LIN {X 59.447,Y -46.624,Z -151.820,A -90.000,B 90.000,C 0.000} C_DIS
LIN {X 59.979,Y -46.636,Z -152.039,A -90.000,B 90.000,C 0.000} C_DIS
LIN {X 60.285,Y -46.643,Z -152.174,A -90.000,B 90.000,C 0.000} C_DIS
LIN {X 60.366,Y -46.645,Z -152.210,A -90.000,B 90.000,C 0.000} C_DIS
LIN {X 60.866,Y -46.657,Z -152.447,A -90.000,B 90.000,C 0.000} C_DIS
LIN {X 60.967,Y -46.654,Z -152.497,A -90.000,B 90.000,C 0.000} C_DIS
LIN {X 61.302,Y -46.635,Z -152.670,A -90.000,B 90.000,C 0.000} C_DIS
LIN {X 61.532,Y -46.619,Z -152.790,A -90.000,B 90.000,C 0.000} C_DIS
LIN {X 62.046,Y -46.587,Z -153.082,A -90.000,B 90.000,C 0.000} C_DIS
LIN {X 62.540,Y -46.557,Z -153.378,A -90.000,B 90.000,C 0.000} C_DIS
LIN {X 63.037,Y -46.527,Z -153.694,A -90.000,B 90.000,C 0.000} C_DIS
LIN {X 63.620,Y -46.494,Z -154.093,A -90.000,B 90.000,C 0.000} C_DIS
LIN {X 63.900,Y -46.478,Z -154.298,A -90.000,B 90.000,C 0.000} C_DIS
LIN {X 64.036,Y -46.460,Z -154.399,A -90.000,B 90.000,C 0.000} C_DIS
LIN {X 64.158,Y -46.443,Z -154.491,A -90.000,B 90.000,C 0.000} C_DIS
LIN {X 64.675,Y -46.369,Z -154.905,A -90.000,B 90.000,C 0.000} C_DIS
LIN {X 65.187,Y -46.297,Z -155.342,A -90.000,B 90.000,C 0.000} C_DIS
LIN {X 65.521,Y -46.250,Z -155.645,A -90.000,B 90.000,C 0.000} C_DIS
LIN {X 66.029,Y -46.178,Z -156.130,A -90.000,B 90.000,C 0.000} C_DIS
LIN {X 66.453,Y -46.120,Z -156.565,A -90.000,B 90.000,C 0.000} C_DIS
LIN {X 66.624,Y -46.096,Z -156.751,A -90.000,B 90.000,C 0.000} C_DIS
LIN {X 66.971,Y -46.029,Z -157.134,A -90.000,B 90.000,C 0.000} C_DIS
LIN {X 67.241,Y -45.966,Z -157.456,A -90.000,B 90.000,C 0.000} C_DIS
LIN {X 67.519,Y -45.898,Z -157.794,A -90.000,B 90.000,C 0.000} C_DIS
LIN {X 67.718,Y -45.848,Z -158.052,A -90.000,B 90.000,C 0.000} C_DIS
LIN {X 68.044,Y -45.766,Z -158.488,A -90.000,B 90.000,C 0.000} C_DIS
LIN {X 68.258,Y -45.712,Z -158.793,A -90.000,B 90.000,C 0.000} C_DIS
LIN {X 68.440,Y -45.666,Z -159.058,A -90.000,B 90.000,C 0.000} C_DIS
LIN {X 68.717,Y -45.595,Z -159.479,A -90.000,B 90.000,C 0.000} C_DIS
LIN {X 68.978,Y -45.527,Z -159.906,A -90.000,B 90.000,C 0.000} C_DIS
LIN {X 69.258,Y -45.454,Z -160.385,A -90.000,B 90.000,C 0.000} C_DIS
LIN {X 69.508,Y -45.387,Z -160.840,A -90.000,B 90.000,C 0.000} C_DIS
LIN {X 69.580,Y -45.368,Z -160.980,A -90.000,B 90.000,C 0.000} C_DIS
LIN {X 69.738,Y -45.308,Z -161.295,A -90.000,B 90.000,C 0.000} C_DIS
LIN {X 69.738,Y -60.000,Z -161.295,A -90.000,B 90.000,C 0.000} C_DIS
LIN {X 51.420,Y -60.000,Z -148.529,A -90.000,B 90.000,C 0.000} C_DIS
LIN {X 51.420,Y -45.308,Z -148.529,A -90.000,B 90.000,C 0.000} C_DIS
LIN {X 51.656,Y -45.359,Z -148.518,A -90.000,B 90.000,C 0.000} C_DIS
LIN {X 52.314,Y -45.502,Z -148.497,A -90.000,B 90.000,C 0.000} C_DIS
LIN {X 52.905,Y -45.633,Z -148.497,A -90.000,B 90.000,C 0.000} C_DIS
LIN {X 53.199,Y -45.699,Z -148.504,A -90.000,B 90.000,C 0.000} C_DIS
LIN {X 53.580,Y -45.759,Z -148.519,A -90.000,B 90.000,C 0.000} C_DIS
LIN {X 54.008,Y -45.829,Z -148.547,A -90.000,B 90.000,C 0.000} C_DIS
LIN {X 54.649,Y -45.936,Z -148.604,A -90.000,B 90.000,C 0.000} C_DIS
LIN {X 55.130,Y -46.016,Z -148.659,A -90.000,B 90.000,C 0.000} C_DIS
LIN {X 55.563,Y -46.087,Z -148.721,A -90.000,B 90.000,C 0.000} C_DIS
LIN {X 55.943,Y -46.141,Z -148.778,A -90.000,B 90.000,C 0.000} C_DIS
LIN {X 56.047,Y -46.155,Z -148.796,A -90.000,B 90.000,C 0.000} C_DIS
LIN {X 56.497,Y -46.195,Z -148.882,A -90.000,B 90.000,C 0.000} C_DIS
LIN {X 56.661,Y -46.209,Z -148.915,A -90.000,B 90.000,C 0.000} C_DIS
LIN {X 57.300,Y -46.275,Z -149.058,A -90.000,B 90.000,C 0.000} C_DIS
LIN {X 57.950,Y -46.344,Z -149.225,A -90.000,B 90.000,C 0.000} C_DIS
LIN {X 58.439,Y -46.397,Z -149.362,A -90.000,B 90.000,C 0.000} C_DIS
LIN {X 58.552,Y -46.409,Z -149.396,A -90.000,B 90.000,C 0.000} C_DIS
LIN {X 58.696,Y -46.417,Z -149.440,A -90.000,B 90.000,C 0.000} C_DIS
LIN {X 59.080,Y -46.425,Z -149.568,A -90.000,B 90.000,C 0.000} C_DIS
LIN {X 59.564,Y -46.434,Z -149.734,A -90.000,B 90.000,C 0.000} C_DIS
LIN {X 59.994,Y -46.444,Z -149.897,A -90.000,B 90.000,C 0.000} C_DIS
LIN {X 60.209,Y -46.450,Z -149.979,A -90.000,B 90.000,C 0.000} C_DIS
LIN {X 60.788,Y -46.470,Z -150.217,A -90.000,B 90.000,C 0.000} C_DIS
LIN {X 61.149,Y -46.483,Z -150.377,A -90.000,B 90.000,C 0.000} C_DIS
LIN {X 61.348,Y -46.491,Z -150.469,A -90.000,B 90.000,C 0.000} C_DIS
LIN {X 61.461,Y -46.494,Z -150.522,A -90.000,B 90.000,C 0.000} C_DIS
LIN {X 61.703,Y -46.490,Z -150.638,A -90.000,B 90.000,C 0.000} C_DIS
LIN {X 61.873,Y -46.482,Z -150.723,A -90.000,B 90.000,C 0.000} C_DIS
LIN {X 62.480,Y -46.449,Z -151.038,A -90.000,B 90.000,C 0.000} C_DIS
LIN {X 63.064,Y -46.419,Z -151.368,A -90.000,B 90.000,C 0.000} C_DIS
LIN {X 63.602,Y -46.393,Z -151.691,A -90.000,B 90.000,C 0.000} C_DIS
LIN {X 64.157,Y -46.368,Z -152.044,A -90.000,B 90.000,C 0.000} C_DIS
LIN {X 64.418,Y -46.358,Z -152.222,A -90.000,B 90.000,C 0.000} C_DIS
LIN {X 64.519,Y -46.351,Z -152.292,A -90.000,B 90.000,C 0.000} C_DIS
LIN {X 64.794,Y -46.316,Z -152.483,A -90.000,B 90.000,C 0.000} C_DIS
LIN {X 65.364,Y -46.243,Z -152.908,A -90.000,B 90.000,C 0.000} C_DIS
LIN {X 65.919,Y -46.170,Z -153.351,A -90.000,B 90.000,C 0.000} C_DIS
LIN {X 66.508,Y -46.088,Z -153.855,A -90.000,B 90.000,C 0.000} C_DIS
LIN {X 66.878,Y -46.036,Z -154.192,A -90.000,B 90.000,C 0.000} C_DIS
LIN {X 67.263,Y -45.983,Z -154.559,A -90.000,B 90.000,C 0.000} C_DIS
LIN {X 67.435,Y -45.949,Z -154.726,A -90.000,B 90.000,C 0.000} C_DIS
LIN {X 67.634,Y -45.911,Z -154.932,A -90.000,B 90.000,C 0.000} C_DIS
LIN {X 67.855,Y -45.862,Z -155.162,A -90.000,B 90.000,C 0.000} C_DIS
LIN {X 68.412,Y -45.738,Z -155.778,A -90.000,B 90.000,C 0.000} C_DIS
LIN {X 68.813,Y -45.649,Z -156.256,A -90.000,B 90.000,C 0.000} C_DIS
LIN {X 69.057,Y -45.594,Z -156.552,A -90.000,B 90.000,C 0.000} C_DIS
LIN {X 69.379,Y -45.522,Z -156.972,A -90.000,B 90.000,C 0.000} C_DIS
LIN {X 69.631,Y -45.465,Z -157.308,A -90.000,B 90.000,C 0.000} C_DIS
LIN {X 69.887,Y -45.407,Z -157.672,A -90.000,B 90.000,C 0.000} C_DIS
LIN {X 70.069,Y -45.363,Z -157.937,A -90.000,B 90.000,C 0.000} C_DIS
LIN {X 70.283,Y -45.308,Z -158.263,A -90.000,B 90.000,C 0.000} C_DIS
LIN {X 70.283,Y -60.000,Z -158.263,A -90.000,B 90.000,C 0.000} C_DIS
LIN {X 53.285,Y -60.000,Z -146.544,A -90.000,B 90.000,C 0.000} C_DIS
LIN {X 53.285,Y -45.308,Z -146.544,A -90.000,B 90.000,C 0.000} C_DIS
LIN {X 53.566,Y -45.372,Z -146.551,A -90.000,B 90.000,C 0.000} C_DIS
LIN {X 53.798,Y -45.420,Z -146.559,A -90.000,B 90.000,C 0.000} C_DIS
LIN {X 53.933,Y -45.449,Z -146.567,A -90.000,B 90.000,C 0.000} C_DIS
LIN {X 54.248,Y -45.505,Z -146.588,A -90.000,B 90.000,C 0.000} C_DIS
LIN {X 54.708,Y -45.588,Z -146.628,A -90.000,B 90.000,C 0.000} C_DIS
LIN {X 54.923,Y -45.624,Z -146.648,A -90.000,B 90.000,C 0.000} C_DIS
LIN {X 55.458,Y -45.716,Z -146.709,A -90.000,B 90.000,C 0.000} C_DIS
LIN {X 56.327,Y -45.869,Z -146.834,A -90.000,B 90.000,C 0.000} C_DIS
LIN {X 56.403,Y -45.881,Z -146.847,A -90.000,B 90.000,C 0.000} C_DIS
LIN {X 56.867,Y -45.935,Z -146.934,A -90.000,B 90.000,C 0.000} C_DIS
LIN {X 57.119,Y -45.961,Z -146.984,A -90.000,B 90.000,C 0.000} C_DIS
LIN {X 57.818,Y -46.036,Z -147.141,A -90.000,B 90.000,C 0.000} C_DIS
LIN {X 58.513,Y -46.115,Z -147.319,A -90.000,B 90.000,C 0.000} C_DIS
LIN {X 59.083,Y -46.192,Z -147.479,A -90.000,B 90.000,C 0.000} C_DIS
LIN {X 59.198,Y -46.208,Z -147.513,A -90.000,B 90.000,C 0.000} C_DIS
LIN {X 59.344,Y -46.218,Z -147.558,A -90.000,B 90.000,C 0.000} C_DIS
LIN {X 59.731,Y -46.232,Z -147.686,A -90.000,B 90.000,C 0.000} C_DIS
LIN {X 60.273,Y -46.252,Z -147.873,A -90.000,B 90.000,C 0.000} C_DIS
LIN {X 60.972,Y -46.281,Z -148.138,A -90.000,B 90.000,C 0.000} C_DIS
LIN {X 61.600,Y -46.310,Z -148.396,A -90.000,B 90.000,C 0.000} C_DIS
LIN {X 61.987,Y -46.328,Z -148.568,A -90.000,B 90.000,C 0.000} C_DIS
LIN {X 62.168,Y -46.329,Z -148.652,A -90.000,B 90.000,C 0.000} C_DIS
LIN {X 62.338,Y -46.325,Z -148.733,A -90.000,B 90.000,C 0.000} C_DIS
LIN {X 62.588,Y -46.314,Z -148.853,A -90.000,B 90.000,C 0.000} C_DIS
LIN {X 62.784,Y -46.305,Z -148.951,A -90.000,B 90.000,C 0.000} C_DIS
LIN {X 62.929,Y -46.298,Z -149.026,A -90.000,B 90.000,C 0.000} C_DIS
LIN {X 63.454,Y -46.274,Z -149.300,A -90.000,B 90.000,C 0.000} C_DIS
LIN {X 64.083,Y -46.246,Z -149.656,A -90.000,B 90.000,C 0.000} C_DIS
LIN {X 64.667,Y -46.221,Z -150.007,A -90.000,B 90.000,C 0.000} C_DIS
LIN {X 65.039,Y -46.205,Z -150.244,A -90.000,B 90.000,C 0.000} C_DIS
LIN {X 65.111,Y -46.200,Z -150.290,A -90.000,B 90.000,C 0.000} C_DIS
LIN {X 65.274,Y -46.179,Z -150.396,A -90.000,B 90.000,C 0.000} C_DIS
LIN {X 65.963,Y -46.090,Z -150.876,A -90.000,B 90.000,C 0.000} C_DIS
LIN {X 66.585,Y -46.011,Z -151.341,A -90.000,B 90.000,C 0.000} C_DIS
LIN {X 67.191,Y -45.937,Z -151.825,A -90.000,B 90.000,C 0.000} C_DIS
LIN {X 67.828,Y -45.860,Z -152.369,A -90.000,B 90.000,C 0.000} C_DIS
LIN {X 68.251,Y -45.787,Z -152.758,A -90.000,B 90.000,C 0.000} C_DIS
LIN {X 68.759,Y -45.683,Z -153.251,A -90.000,B 90.000,C 0.000} C_DIS
LIN {X 68.852,Y -45.664,Z -153.343,A -90.000,B 90.000,C 0.000} C_DIS
LIN {X 69.222,Y -45.588,Z -153.728,A -90.000,B 90.000,C 0.000} C_DIS
LIN {X 69.305,Y -45.570,Z -153.815,A -90.000,B 90.000,C 0.000} C_DIS
LIN {X 69.898,Y -45.438,Z -154.474,A -90.000,B 90.000,C 0.000} C_DIS
LIN {X 70.312,Y -45.346,Z -154.966,A -90.000,B 90.000,C 0.000} C_DIS
LIN {X 70.480,Y -45.308,Z -155.171,A -90.000,B 90.000,C 0.000} C_DIS
LIN {X 70.480,Y -60.000,Z -155.171,A -90.000,B 90.000,C 0.000} C_DIS
LIN {X 55.397,Y -60.000,Z -144.721,A -90.000,B 90.000,C 0.000} C_DIS
LIN {X 55.397,Y -45.308,Z -144.721,A -90.000,B 90.000,C 0.000} C_DIS
LIN {X 55.811,Y -45.386,Z -144.768,A -90.000,B 90.000,C 0.000} C_DIS
LIN {X 56.720,Y -45.560,Z -144.897,A -90.000,B 90.000,C 0.000} C_DIS
LIN {X 57.059,Y -45.621,Z -144.957,A -90.000,B 90.000,C 0.000} C_DIS
LIN {X 57.528,Y -45.677,Z -145.047,A -90.000,B 90.000,C 0.000} C_DIS
LIN {X 57.647,Y -45.689,Z -145.073,A -90.000,B 90.000,C 0.000} C_DIS
LIN {X 58.339,Y -45.777,Z -145.227,A -90.000,B 90.000,C 0.000} C_DIS
LIN {X 59.096,Y -45.878,Z -145.421,A -90.000,B 90.000,C 0.000} C_DIS
LIN {X 59.727,Y -45.963,Z -145.598,A -90.000,B 90.000,C 0.000} C_DIS
LIN {X 59.823,Y -45.976,Z -145.627,A -90.000,B 90.000,C 0.000} C_DIS
LIN {X 59.969,Y -45.987,Z -145.672,A -90.000,B 90.000,C 0.000} C_DIS
LIN {X 60.421,Y -46.003,Z -145.823,A -90.000,B 90.000,C 0.000} C_DIS
LIN {X 60.636,Y -46.011,Z -145.897,A -90.000,B 90.000,C 0.000} C_DIS
LIN {X 60.986,Y -46.030,Z -146.017,A -90.000,B 90.000,C 0.000} C_DIS
LIN {X 61.738,Y -46.074,Z -146.302,A -90.000,B 90.000,C 0.000} C_DIS
LIN {X 62.412,Y -46.116,Z -146.579,A -90.000,B 90.000,C 0.000} C_DIS
LIN {X 62.556,Y -46.122,Z -146.643,A -90.000,B 90.000,C 0.000} C_DIS
LIN {X 62.721,Y -46.124,Z -146.716,A -90.000,B 90.000,C 0.000} C_DIS
LIN {X 62.878,Y -46.121,Z -146.788,A -90.000,B 90.000,C 0.000} C_DIS
LIN {X 63.515,Y -46.097,Z -147.094,A -90.000,B 90.000,C 0.000} C_DIS
LIN {X 63.692,Y -46.091,Z -147.182,A -90.000,B 90.000,C 0.000} C_DIS
LIN {X 64.428,Y -46.066,Z -147.565,A -90.000,B 90.000,C 0.000} C_DIS
LIN {X 65.103,Y -46.053,Z -147.946,A -90.000,B 90.000,C 0.000} C_DIS
LIN {X 65.440,Y -46.047,Z -148.148,A -90.000,B 90.000,C 0.000} C_DIS
LIN {X 65.570,Y -46.042,Z -148.226,A -90.000,B 90.000,C 0.000} C_DIS
LIN {X 65.702,Y -46.029,Z -148.306,A -90.000,B 90.000,C 0.000} C_DIS
LIN {X 66.341,Y -45.956,Z -148.719,A -90.000,B 90.000,C 0.000} C_DIS
LIN {X 67.136,Y -45.868,Z -149.271,A -90.000,B 90.000,C 0.000} C_DIS
LIN {X 67.565,Y -45.821,Z -149.592,A -90.000,B 90.000,C 0.000} C_DIS
LIN {X 67.809,Y -45.791,Z -149.775,A -90.000,B 90.000,C 0.000} C_DIS
LIN {X 68.439,Y -45.713,Z -150.279,A -90.000,B 90.000,C 0.000} C_DIS
LIN {X 68.852,Y -45.639,Z -150.635,A -90.000,B 90.000,C 0.000} C_DIS
LIN {X 69.142,Y -45.580,Z -150.888,A -90.000,B 90.000,C 0.000} C_DIS
LIN {X 69.595,Y -45.487,Z -151.308,A -90.000,B 90.000,C 0.000} C_DIS
LIN {X 70.122,Y -45.379,Z -151.819,A -90.000,B 90.000,C 0.000} C_DIS
LIN {X 70.295,Y -45.344,Z -151.995,A -90.000,B 90.000,C 0.000} C_DIS
LIN {X 70.471,Y -45.308,Z -152.177,A -90.000,B 90.000,C 0.000} C_DIS
LIN {X 70.471,Y -60.000,Z -152.177,A -90.000,B 90.000,C 0.000} C_DIS
LIN {X 57.673,Y -60.000,Z -143.068,A -90.000,B 90.000,C 0.000} C_DIS
LIN {X 57.673,Y -45.308,Z -143.068,A -90.000,B 90.000,C 0.000} C_DIS
LIN {X 57.981,Y -45.358,Z -143.125,A -90.000,B 90.000,C 0.000} C_DIS
LIN {X 58.562,Y -45.455,Z -143.250,A -90.000,B 90.000,C 0.000} C_DIS
LIN {X 58.857,Y -45.494,Z -143.316,A -90.000,B 90.000,C 0.000} C_DIS
LIN {X 59.667,Y -45.605,Z -143.524,A -90.000,B 90.000,C 0.000} C_DIS
LIN {X 60.166,Y -45.674,Z -143.664,A -90.000,B 90.000,C 0.000} C_DIS
LIN {X 60.407,Y -45.704,Z -143.734,A -90.000,B 90.000,C 0.000} C_DIS
LIN {X 60.688,Y -45.731,Z -143.821,A -90.000,B 90.000,C 0.000} C_DIS
LIN {X 61.226,Y -45.785,Z -143.998,A -90.000,B 90.000,C 0.000} C_DIS
LIN {X 61.701,Y -45.815,Z -144.162,A -90.000,B 90.000,C 0.000} C_DIS
LIN {X 62.505,Y -45.867,Z -144.467,A -90.000,B 90.000,C 0.000} C_DIS
LIN {X 62.948,Y -45.898,Z -144.648,A -90.000,B 90.000,C 0.000} C_DIS
LIN {X 63.151,Y -45.907,Z -144.732,A -90.000,B 90.000,C 0.000} C_DIS
LIN {X 63.524,Y -45.912,Z -144.897,A -90.000,B 90.000,C 0.000} C_DIS
LIN {X 63.817,Y -45.906,Z -145.033,A -90.000,B 90.000,C 0.000} C_DIS
LIN {X 64.402,Y -45.896,Z -145.312,A -90.000,B 90.000,C 0.000} C_DIS
LIN {X 64.615,Y -45.892,Z -145.419,A -90.000,B 90.000,C 0.000} C_DIS
LIN {X 65.404,Y -45.875,Z -145.830,A -90.000,B 90.000,C 0.000} C_DIS
LIN {X 65.989,Y -45.864,Z -146.160,A -90.000,B 90.000,C 0.000} C_DIS
LIN {X 66.114,Y -45.858,Z -146.231,A -90.000,B 90.000,C 0.000} C_DIS
LIN {X 66.199,Y -45.850,Z -146.283,A -90.000,B 90.000,C 0.000} C_DIS
LIN {X 66.754,Y -45.786,Z -146.623,A -90.000,B 90.000,C 0.000} C_DIS
LIN {X 67.454,Y -45.711,Z -147.076,A -90.000,B 90.000,C 0.000} C_DIS
LIN {X 67.702,Y -45.686,Z -147.248,A -90.000,B 90.000,C 0.000} C_DIS
LIN {X 68.305,Y -45.623,Z -147.667,A -90.000,B 90.000,C 0.000} C_DIS
LIN {X 68.893,Y -45.563,Z -148.106,A -90.000,B 90.000,C 0.000} C_DIS
LIN {X 69.052,Y -45.538,Z -148.229,A -90.000,B 90.000,C 0.000} C_DIS
LIN {X 69.317,Y -45.495,Z -148.442,A -90.000,B 90.000,C 0.000} C_DIS
LIN {X 69.700,Y -45.422,Z -148.754,A -90.000,B 90.000,C 0.000} C_DIS
LIN {X 70.298,Y -45.308,Z -149.272,A -90.000,B 90.000,C 0.000} C_DIS
LIN {X 70.298,Y -60.000,Z -149.272,A -90.000,B 90.000,C 0.000} C_DIS
LIN {X 60.225,Y -60.000,Z -141.626,A -90.000,B 90.000,C 0.000} C_DIS
LIN {X 60.225,Y -45.308,Z -141.626,A -90.000,B 90.000,C 0.000} C_DIS
LIN {X 60.347,Y -45.329,Z -141.660,A -90.000,B 90.000,C 0.000} C_DIS
LIN {X 60.767,Y -45.387,Z -141.778,A -90.000,B 90.000,C 0.000} C_DIS
LIN {X 60.971,Y -45.412,Z -141.837,A -90.000,B 90.000,C 0.000} C_DIS
LIN {X 61.330,Y -45.447,Z -141.949,A -90.000,B 90.000,C 0.000} C_DIS
LIN {X 61.949,Y -45.509,Z -142.153,A -90.000,B 90.000,C 0.000} C_DIS
LIN {X 62.419,Y -45.557,Z -142.313,A -90.000,B 90.000,C 0.000} C_DIS
LIN {X 62.933,Y -45.611,Z -142.505,A -90.000,B 90.000,C 0.000} C_DIS
LIN {X 63.273,Y -45.634,Z -142.635,A -90.000,B 90.000,C 0.000} C_DIS
LIN {X 63.488,Y -45.648,Z -142.723,A -90.000,B 90.000,C 0.000} C_DIS
LIN {X 63.608,Y -45.654,Z -142.773,A -90.000,B 90.000,C 0.000} C_DIS
LIN {X 63.900,Y -45.658,Z -142.895,A -90.000,B 90.000,C 0.000} C_DIS
LIN {X 64.355,Y -45.665,Z -143.095,A -90.000,B 90.000,C 0.000} C_DIS
LIN {X 64.669,Y -45.670,Z -143.239,A -90.000,B 90.000,C 0.000} C_DIS
LIN {X 65.147,Y -45.679,Z -143.465,A -90.000,B 90.000,C 0.000} C_DIS
LIN {X 65.384,Y -45.675,Z -143.581,A -90.000,B 90.000,C 0.000} C_DIS
LIN {X 65.531,Y -45.673,Z -143.654,A -90.000,B 90.000,C 0.000} C_DIS
LIN {X 66.367,Y -45.661,Z -144.090,A -90.000,B 90.000,C 0.000} C_DIS
LIN {X 66.431,Y -45.660,Z -144.126,A -90.000,B 90.000,C 0.000} C_DIS
LIN {X 66.624,Y -45.649,Z -144.236,A -90.000,B 90.000,C 0.000} C_DIS
LIN {X 67.126,Y -45.612,Z -144.524,A -90.000,B 90.000,C 0.000} C_DIS
LIN {X 67.404,Y -45.592,Z -144.692,A -90.000,B 90.000,C 0.000} C_DIS
LIN {X 67.816,Y -45.551,Z -144.944,A -90.000,B 90.000,C 0.000} C_DIS
LIN {X 68.570,Y -45.476,Z -145.433,A -90.000,B 90.000,C 0.000} C_DIS
LIN {X 69.377,Y -45.399,Z -145.993,A -90.000,B 90.000,C 0.000} C_DIS
LIN {X 69.423,Y -45.392,Z -146.025,A -90.000,B 90.000,C 0.000} C_DIS
LIN {X 69.561,Y -45.372,Z -146.127,A -90.000,B 90.000,C 0.000} C_DIS
LIN {X 69.817,Y -45.330,Z -146.321,A -90.000,B 90.000,C 0.000} C_DIS
LIN {X 69.929,Y -45.308,Z -146.406,A -90.000,B 90.000,C 0.000} C_DIS
LIN {X 70.238,Y -45.253,Z -146.643,A -90.000,B 90.000,C 0.000} C_DIS
LIN {X 70.507,Y -45.203,Z -146.852,A -90.000,B 90.000,C 0.000} C_DIS
LIN {X 70.735,Y -45.160,Z -147.034,A -90.000,B 90.000,C 0.000} C_DIS
LIN {X 71.005,Y -45.110,Z -147.258,A -90.000,B 90.000,C 0.000} C_DIS
LIN {X 71.139,Y -45.085,Z -147.375,A -90.000,B 90.000,C 0.000} C_DIS
LIN {X 71.274,Y -45.060,Z -147.506,A -90.000,B 90.000,C 0.000} C_DIS
LIN {X 71.302,Y -45.055,Z -147.538,A -90.000,B 90.000,C 0.000} C_DIS
LIN {X 71.330,Y -45.050,Z -147.575,A -90.000,B 90.000,C 0.000} C_DIS
LIN {X 71.338,Y -45.049,Z -147.593,A -90.000,B 90.000,C 0.000} C_DIS
LIN {X 71.339,Y -45.049,Z -147.600,A -90.000,B 90.000,C 0.000} C_DIS
LIN {X 71.336,Y -45.049,Z -147.610,A -90.000,B 90.000,C 0.000} C_DIS
LIN {X 71.317,Y -45.053,Z -147.616,A -90.000,B 90.000,C 0.000} C_DIS
LIN {X 71.282,Y -45.061,Z -147.610,A -90.000,B 90.000,C 0.000} C_DIS
LIN {X 71.250,Y -45.067,Z -147.599,A -90.000,B 90.000,C 0.000} C_DIS
LIN {X 71.166,Y -45.084,Z -147.565,A -90.000,B 90.000,C 0.000} C_DIS
LIN {X 70.992,Y -45.117,Z -147.479,A -90.000,B 90.000,C 0.000} C_DIS
LIN {X 70.677,Y -45.178,Z -147.305,A -90.000,B 90.000,C 0.000} C_DIS
LIN {X 70.279,Y -45.255,Z -147.070,A -90.000,B 90.000,C 0.000} C_DIS
LIN {X 69.809,Y -45.347,Z -146.780,A -90.000,B 90.000,C 0.000} C_DIS
LIN {X 69.550,Y -45.397,Z -146.617,A -90.000,B 90.000,C 0.000} C_DIS
LIN {X 69.276,Y -45.435,Z -146.443,A -90.000,B 90.000,C 0.000} C_DIS
LIN {X 68.693,Y -45.497,Z -146.065,A -90.000,B 90.000,C 0.000} C_DIS
LIN {X 68.386,Y -45.528,Z -145.863,A -90.000,B 90.000,C 0.000} C_DIS
LIN {X 67.747,Y -45.591,Z -145.437,A -90.000,B 90.000,C 0.000} C_DIS
LIN {X 67.084,Y -45.654,Z -144.987,A -90.000,B 90.000,C 0.000} C_DIS
LIN {X 66.409,Y -45.696,Z -144.520,A -90.000,B 90.000,C 0.000} C_DIS
LIN {X 66.070,Y -45.699,Z -144.283,A -90.000,B 90.000,C 0.000} C_DIS
LIN {X 65.396,Y -45.697,Z -143.804,A -90.000,B 90.000,C 0.000} C_DIS
LIN {X 65.065,Y -45.695,Z -143.564,A -90.000,B 90.000,C 0.000} C_DIS
LIN {X 64.738,Y -45.679,Z -143.325,A -90.000,B 90.000,C 0.000} C_DIS
LIN {X 64.105,Y -45.646,Z -142.853,A -90.000,B 90.000,C 0.000} C_DIS
LIN {X 63.801,Y -45.629,Z -142.622,A -90.000,B 90.000,C 0.000} C_DIS
LIN {X 63.508,Y -45.605,Z -142.396,A -90.000,B 90.000,C 0.000} C_DIS
LIN {X 63.227,Y -45.571,Z -142.174,A -90.000,B 90.000,C 0.000} C_DIS
LIN {X 62.959,Y -45.526,Z -141.959,A -90.000,B 90.000,C 0.000} C_DIS
LIN {X 62.585,Y -45.457,Z -141.649,A -90.000,B 90.000,C 0.000} C_DIS
LIN {X 62.249,Y -45.398,Z -141.357,A -90.000,B 90.000,C 0.000} C_DIS
LIN {X 62.048,Y -45.361,Z -141.175,A -90.000,B 90.000,C 0.000} C_DIS
LIN {X 61.867,Y -45.327,Z -141.003,A -90.000,B 90.000,C 0.000} C_DIS
LIN {X 61.707,Y -45.294,Z -140.842,A -90.000,B 90.000,C 0.000} C_DIS
LIN {X 61.571,Y -45.257,Z -140.692,A -90.000,B 90.000,C 0.000} C_DIS
LIN {X 61.458,Y -45.222,Z -140.556,A -90.000,B 90.000,C 0.000} C_DIS
LIN {X 61.411,Y -45.206,Z -140.493,A -90.000,B 90.000,C 0.000} C_DIS
LIN {X 61.371,Y -45.191,Z -140.434,A -90.000,B 90.000,C 0.000} C_DIS
LIN {X 61.324,Y -45.172,Z -140.352,A -90.000,B 90.000,C 0.000} C_DIS
LIN {X 61.292,Y -45.155,Z -140.278,A -90.000,B 90.000,C 0.000} C_DIS
LIN {X 61.280,Y -45.146,Z -140.234,A -90.000,B 90.000,C 0.000} C_DIS
LIN {X 61.275,Y -45.134,Z -140.175,A -90.000,B 90.000,C 0.000} C_DIS
LIN {X 61.282,Y -45.129,Z -140.142,A -90.000,B 90.000,C 0.000} C_DIS
LIN {X 61.296,Y -45.124,Z -140.112,A -90.000,B 90.000,C 0.000} C_DIS
LIN {X 61.307,Y -45.123,Z -140.099,A -90.000,B 90.000,C 0.000} C_DIS
LIN {X 61.333,Y -45.120,Z -140.076,A -90.000,B 90.000,C 0.000} C_DIS
LIN {X 61.389,Y -45.120,Z -140.051,A -90.000,B 90.000,C 0.000} C_DIS
LIN {X 61.436,Y -45.122,Z -140.040,A -90.000,B 90.000,C 0.000} C_DIS
LIN {X 61.492,Y -45.125,Z -140.034,A -90.000,B 90.000,C 0.000} C_DIS
LIN {X 61.558,Y -45.130,Z -140.033,A -90.000,B 90.000,C 0.000} C_DIS
LIN {X 61.672,Y -45.141,Z -140.041,A -90.000,B 90.000,C 0.000} C_DIS
LIN {X 61.760,Y -45.151,Z -140.053,A -90.000,B 90.000,C 0.000} C_DIS
LIN {X 61.965,Y -45.175,Z -140.093,A -90.000,B 90.000,C 0.000} C_DIS
LIN {X 62.209,Y -45.207,Z -140.155,A -90.000,B 90.000,C 0.000} C_DIS
LIN {X 62.346,Y -45.225,Z -140.195,A -90.000,B 90.000,C 0.000} C_DIS
LIN {X 62.494,Y -45.241,Z -140.240,A -90.000,B 90.000,C 0.000} C_DIS
LIN {X 62.820,Y -45.272,Z -140.349,A -90.000,B 90.000,C 0.000} C_DIS
LIN {X 63.190,Y -45.308,Z -140.484,A -90.000,B 90.000,C 0.000} C_DIS
LIN {X 63.862,Y -45.376,Z -140.736,A -90.000,B 90.000,C 0.000} C_DIS
LIN {X 63.917,Y -45.381,Z -140.756,A -90.000,B 90.000,C 0.000} C_DIS
LIN {X 64.135,Y -45.392,Z -140.844,A -90.000,B 90.000,C 0.000} C_DIS
LIN {X 64.700,Y -45.422,Z -141.077,A -90.000,B 90.000,C 0.000} C_DIS
LIN {X 65.187,Y -45.427,Z -141.292,A -90.000,B 90.000,C 0.000} C_DIS
LIN {X 65.574,Y -45.432,Z -141.470,A -90.000,B 90.000,C 0.000} C_DIS
LIN {X 66.014,Y -45.438,Z -141.679,A -90.000,B 90.000,C 0.000} C_DIS
LIN {X 66.418,Y -45.444,Z -141.876,A -90.000,B 90.000,C 0.000} C_DIS
LIN {X 66.710,Y -45.449,Z -142.027,A -90.000,B 90.000,C 0.000} C_DIS
LIN {X 66.868,Y -45.447,Z -142.109,A -90.000,B 90.000,C 0.000} C_DIS
LIN {X 67.087,Y -45.434,Z -142.225,A -90.000,B 90.000,C 0.000} C_DIS
LIN {X 67.353,Y -45.413,Z -142.368,A -90.000,B 90.000,C 0.000} C_DIS
LIN {X 68.139,Y -45.355,Z -142.819,A -90.000,B 90.000,C 0.000} C_DIS
LIN {X 68.795,Y -45.308,Z -143.217,A -90.000,B 90.000,C 0.000} C_DIS
LIN {X 68.795,Y -60.000,Z -143.217,A -90.000,B 90.000,C 0.000} C_DIS
LIN {X 21.437,Y -60.000,Z -200.643,A -90.000,B 90.000,C 0.000} C_DIS
LIN {X 21.437,Y -45.308,Z -200.643,A -90.000,B 90.000,C 0.000} C_DIS
LIN {X 21.642,Y -45.328,Z -200.052,A -90.000,B 90.000,C 0.000} C_DIS
LIN {X 21.753,Y -45.340,Z -199.753,A -90.000,B 90.000,C 0.000} C_DIS
LIN {X 22.022,Y -45.372,Z -199.088,A -90.000,B 90.000,C 0.000} C_DIS
LIN {X 22.066,Y -45.377,Z -198.962,A -90.000,B 90.000,C 0.000} C_DIS
LIN {X 22.972,Y -45.479,Z -196.594,A -90.000,B 90.000,C 0.000} C_DIS
LIN {X 23.048,Y -45.481,Z -196.226,A -90.000,B 90.000,C 0.000} C_DIS
LIN {X 23.142,Y -45.482,Z -195.852,A -90.000,B 90.000,C 0.000} C_DIS
LIN {X 23.197,Y -45.483,Z -195.651,A -90.000,B 90.000,C 0.000} C_DIS
LIN {X 23.294,Y -45.486,Z -195.320,A -90.000,B 90.000,C 0.000} C_DIS
LIN {X 23.416,Y -45.489,Z -194.956,A -90.000,B 90.000,C 0.000} C_DIS
LIN {X 23.860,Y -45.511,Z -193.771,A -90.000,B 90.000,C 0.000} C_DIS
LIN {X 23.928,Y -45.489,Z -193.299,A -90.000,B 90.000,C 0.000} C_DIS
LIN {X 23.996,Y -45.472,Z -192.905,A -90.000,B 90.000,C 0.000} C_DIS
LIN {X 24.063,Y -45.462,Z -192.583,A -90.000,B 90.000,C 0.000} C_DIS
LIN {X 24.148,Y -45.454,Z -192.215,A -90.000,B 90.000,C 0.000} C_DIS
LIN {X 24.221,Y -45.442,Z -191.941,A -90.000,B 90.000,C 0.000} C_DIS
LIN {X 24.335,Y -45.426,Z -191.571,A -90.000,B 90.000,C 0.000} C_DIS
LIN {X 24.388,Y -45.420,Z -191.413,A -90.000,B 90.000,C 0.000} C_DIS
LIN {X 24.556,Y -45.407,Z -190.951,A -90.000,B 90.000,C 0.000} C_DIS
LIN {X 24.669,Y -45.402,Z -190.671,A -90.000,B 90.000,C 0.000} C_DIS
LIN {X 24.849,Y -45.402,Z -190.259,A -90.000,B 90.000,C 0.000} C_DIS
LIN {X 24.895,Y -45.402,Z -190.152,A -90.000,B 90.000,C 0.000} C_DIS
LIN {X 25.316,Y -45.322,Z -188.533,A -90.000,B 90.000,C 0.000} C_DIS
LIN {X 25.368,Y -45.315,Z -188.359,A -90.000,B 90.000,C 0.000} C_DIS
LIN {X 25.390,Y -45.308,Z -188.285,A -90.000,B 90.000,C 0.000} C_DIS
LIN {X 25.390,Y -60.000,Z -188.285,A -90.000,B 90.000,C 0.000} C_DIS
LIN {X 9.368,Y -60.000,Z -243.561,A -90.000,B 90.000,C 0.000} C_DIS
LIN {X 9.368,Y -46.616,Z -243.561,A -90.000,B 90.000,C 0.000} C_DIS
LIN {X 8.562,Y -46.555,Z -242.196,A -90.000,B 90.000,C 0.000} C_DIS
LIN {X 8.317,Y -46.536,Z -241.760,A -90.000,B 90.000,C 0.000} C_DIS
LIN {X 8.219,Y -46.529,Z -241.573,A -90.000,B 90.000,C 0.000} C_DIS
LIN {X 8.140,Y -46.518,Z -241.417,A -90.000,B 90.000,C 0.000} C_DIS
LIN {X 7.998,Y -46.498,Z -241.118,A -90.000,B 90.000,C 0.000} C_DIS
LIN {X 7.944,Y -46.481,Z -240.992,A -90.000,B 90.000,C 0.000} C_DIS
LIN {X 7.869,Y -46.458,Z -240.814,A -90.000,B 90.000,C 0.000} C_DIS
LIN {X 7.812,Y -46.439,Z -240.672,A -90.000,B 90.000,C 0.000} C_DIS
LIN {X 7.699,Y -46.399,Z -240.353,A -90.000,B 90.000,C 0.000} C_DIS
LIN {X 7.516,Y -46.327,Z -239.759,A -90.000,B 90.000,C 0.000} C_DIS
LIN {X 7.433,Y -46.294,Z -239.471,A -90.000,B 90.000,C 0.000} C_DIS
LIN {X 7.370,Y -46.266,Z -239.217,A -90.000,B 90.000,C 0.000} C_DIS
LIN {X 7.341,Y -46.252,Z -239.092,A -90.000,B 90.000,C 0.000} C_DIS
LIN {X 7.280,Y -46.220,Z -238.781,A -90.000,B 90.000,C 0.000} C_DIS
LIN {X 7.237,Y -46.193,Z -238.516,A -90.000,B 90.000,C 0.000} C_DIS
LIN {X 7.145,Y -46.124,Z -237.812,A -90.000,B 90.000,C 0.000} C_DIS
LIN {X 7.104,Y -46.084,Z -237.389,A -90.000,B 90.000,C 0.000} C_DIS
LIN {X 7.085,Y -46.059,Z -237.120,A -90.000,B 90.000,C 0.000} C_DIS
LIN {X 7.067,Y -46.020,Z -236.662,A -90.000,B 90.000,C 0.000} C_DIS
LIN {X 7.065,Y -46.009,Z -236.537,A -90.000,B 90.000,C 0.000} C_DIS
LIN {X 7.066,Y -45.986,Z -236.300,A -90.000,B 90.000,C 0.000} C_DIS
LIN {X 7.070,Y -45.967,Z -236.107,A -90.000,B 90.000,C 0.000} C_DIS
LIN {X 7.087,Y -45.932,Z -235.742,A -90.000,B 90.000,C 0.000} C_DIS
LIN {X 7.111,Y -45.901,Z -235.468,A -90.000,B 90.000,C 0.000} C_DIS
LIN {X 7.143,Y -45.872,Z -235.204,A -90.000,B 90.000,C 0.000} C_DIS
LIN {X 7.175,Y -45.848,Z -234.971,A -90.000,B 90.000,C 0.000} C_DIS
LIN {X 7.243,Y -45.810,Z -234.578,A -90.000,B 90.000,C 0.000} C_DIS
LIN {X 7.485,Y -45.705,Z -233.428,A -90.000,B 90.000,C 0.000} C_DIS
LIN {X 8.325,Y -45.354,Z -229.481,A -90.000,B 90.000,C 0.000} C_DIS
LIN {X 8.459,Y -45.308,Z -228.933,A -90.000,B 90.000,C 0.000} C_DIS
LIN {X 8.459,Y -60.000,Z -228.933,A -90.000,B 90.000,C 0.000} C_DIS
LIN {X 7.048,Y -60.000,Z -243.561,A -90.000,B 90.000,C 0.000} C_DIS
LIN {X 7.048,Y -46.480,Z -243.561,A -90.000,B 90.000,C 0.000} C_DIS
LIN {X 6.824,Y -46.464,Z -243.180,A -90.000,B 90.000,C 0.000} C_DIS
LIN {X 6.581,Y -46.432,Z -242.748,A -90.000,B 90.000,C 0.000} C_DIS
LIN {X 6.545,Y -46.422,Z -242.681,A -90.000,B 90.000,C 0.000} C_DIS
LIN {X 6.339,Y -46.363,Z -242.273,A -90.000,B 90.000,C 0.000} C_DIS
LIN {X 6.202,Y -46.321,Z -241.980,A -90.000,B 90.000,C 0.000} C_DIS
LIN {X 6.124,Y -46.297,Z -241.802,A -90.000,B 90.000,C 0.000} C_DIS
LIN {X 5.973,Y -46.248,Z -241.435,A -90.000,B 90.000,C 0.000} C_DIS
LIN {X 5.831,Y -46.198,Z -241.039,A -90.000,B 90.000,C 0.000} C_DIS
LIN {X 5.774,Y -46.176,Z -240.860,A -90.000,B 90.000,C 0.000} C_DIS
LIN {X 5.623,Y -46.126,Z -240.373,A -90.000,B 90.000,C 0.000} C_DIS
LIN {X 5.524,Y -46.091,Z -240.032,A -90.000,B 90.000,C 0.000} C_DIS
LIN {X 5.445,Y -46.060,Z -239.719,A -90.000,B 90.000,C 0.000} C_DIS
LIN {X 5.414,Y -46.047,Z -239.587,A -90.000,B 90.000,C 0.000} C_DIS
LIN {X 5.333,Y -46.010,Z -239.188,A -90.000,B 90.000,C 0.000} C_DIS
LIN {X 5.277,Y -45.980,Z -238.856,A -90.000,B 90.000,C 0.000} C_DIS
LIN {X 5.242,Y -45.957,Z -238.595,A -90.000,B 90.000,C 0.000} C_DIS
LIN {X 5.179,Y -45.886,Z -238.090,A -90.000,B 90.000,C 0.000} C_DIS
LIN {X 5.134,Y -45.817,Z -237.606,A -90.000,B 90.000,C 0.000} C_DIS
LIN {X 5.119,Y -45.786,Z -237.386,A -90.000,B 90.000,C 0.000} C_DIS
LIN {X 5.109,Y -45.761,Z -237.197,A -90.000,B 90.000,C 0.000} C_DIS
LIN {X 5.093,Y -45.689,Z -236.657,A -90.000,B 90.000,C 0.000} C_DIS
LIN {X 5.095,Y -45.647,Z -236.324,A -90.000,B 90.000,C 0.000} C_DIS
LIN {X 5.103,Y -45.614,Z -236.053,A -90.000,B 90.000,C 0.000} C_DIS
LIN {X 5.126,Y -45.561,Z -235.614,A -90.000,B 90.000,C 0.000} C_DIS
LIN {X 5.152,Y -45.527,Z -235.321,A -90.000,B 90.000,C 0.000} C_DIS
LIN {X 5.188,Y -45.493,Z -235.012,A -90.000,B 90.000,C 0.000} C_DIS
LIN {X 5.226,Y -45.464,Z -234.741,A -90.000,B 90.000,C 0.000} C_DIS
LIN {X 5.305,Y -45.418,Z -234.280,A -90.000,B 90.000,C 0.000} C_DIS
LIN {X 5.544,Y -45.308,Z -233.142,A -90.000,B 90.000,C 0.000} C_DIS
LIN {X 5.544,Y -60.000,Z -233.142,A -90.000,B 90.000,C 0.000} C_DIS
LIN {X 4.754,Y -60.000,Z -243.561,A -90.000,B 90.000,C 0.000} C_DIS
LIN {X 4.754,Y -46.292,Z -243.561,A -90.000,B 90.000,C 0.000} C_DIS
LIN {X 4.565,Y -46.240,Z -243.188,A -90.000,B 90.000,C 0.000} C_DIS
LIN {X 4.400,Y -46.198,Z -242.838,A -90.000,B 90.000,C 0.000} C_DIS
LIN {X 4.339,Y -46.183,Z -242.701,A -90.000,B 90.000,C 0.000} C_DIS
LIN {X 4.133,Y -46.127,Z -242.209,A -90.000,B 90.000,C 0.000} C_DIS
LIN {X 4.099,Y -46.117,Z -242.122,A -90.000,B 90.000,C 0.000} C_DIS
LIN {X 3.934,Y -46.067,Z -241.658,A -90.000,B 90.000,C 0.000} C_DIS
LIN {X 3.732,Y -46.001,Z -241.013,A -90.000,B 90.000,C 0.000} C_DIS
LIN {X 3.611,Y -45.958,Z -240.600,A -90.000,B 90.000,C 0.000} C_DIS
LIN {X 3.572,Y -45.944,Z -240.449,A -90.000,B 90.000,C 0.000} C_DIS
LIN {X 3.535,Y -45.920,Z -240.300,A -90.000,B 90.000,C 0.000} C_DIS
LIN {X 3.475,Y -45.879,Z -240.045,A -90.000,B 90.000,C 0.000} C_DIS
LIN {X 3.387,Y -45.810,Z -239.603,A -90.000,B 90.000,C 0.000} C_DIS
LIN {X 3.321,Y -45.749,Z -239.205,A -90.000,B 90.000,C 0.000} C_DIS
LIN {X 3.216,Y -45.626,Z -238.372,A -90.000,B 90.000,C 0.000} C_DIS
LIN {X 3.164,Y -45.548,Z -237.829,A -90.000,B 90.000,C 0.000} C_DIS
LIN {X 3.145,Y -45.510,Z -237.559,A -90.000,B 90.000,C 0.000} C_DIS
LIN {X 3.134,Y -45.481,Z -237.343,A -90.000,B 90.000,C 0.000} C_DIS
LIN {X 3.116,Y -45.402,Z -236.750,A -90.000,B 90.000,C 0.000} C_DIS
LIN {X 3.117,Y -45.355,Z -236.391,A -90.000,B 90.000,C 0.000} C_DIS
LIN {X 3.126,Y -45.308,Z -236.012,A -90.000,B 90.000,C 0.000} C_DIS
LIN {X 3.129,Y -45.292,Z -235.840,A -90.000,B 90.000,C 0.000} C_DIS
LIN {X 3.148,Y -45.237,Z -235.389,A -90.000,B 90.000,C 0.000} C_DIS
LIN {X 3.163,Y -45.207,Z -235.139,A -90.000,B 90.000,C 0.000} C_DIS
LIN {X 3.191,Y -45.167,Z -234.837,A -90.000,B 90.000,C 0.000} C_DIS
LIN {X 3.212,Y -45.147,Z -234.683,A -90.000,B 90.000,C 0.000} C_DIS
LIN {X 3.223,Y -45.139,Z -234.619,A -90.000,B 90.000,C 0.000} C_DIS
LIN {X 3.247,Y -45.128,Z -234.519,A -90.000,B 90.000,C 0.000} C_DIS
LIN {X 3.258,Y -45.124,Z -234.480,A -90.000,B 90.000,C 0.000} C_DIS
LIN {X 3.278,Y -45.121,Z -234.440,A -90.000,B 90.000,C 0.000} C_DIS
LIN {X 3.292,Y -45.121,Z -234.423,A -90.000,B 90.000,C 0.000} C_DIS
LIN {X 3.311,Y -45.123,Z -234.413,A -90.000,B 90.000,C 0.000} C_DIS
LIN {X 3.326,Y -45.126,Z -234.416,A -90.000,B 90.000,C 0.000} C_DIS
LIN {X 3.348,Y -45.133,Z -234.434,A -90.000,B 90.000,C 0.000} C_DIS
LIN {X 3.385,Y -45.150,Z -234.500,A -90.000,B 90.000,C 0.000} C_DIS
LIN {X 3.401,Y -45.159,Z -234.539,A -90.000,B 90.000,C 0.000} C_DIS
LIN {X 3.432,Y -45.180,Z -234.636,A -90.000,B 90.000,C 0.000} C_DIS
LIN {X 3.465,Y -45.204,Z -234.758,A -90.000,B 90.000,C 0.000} C_DIS
LIN {X 3.516,Y -45.242,Z -234.985,A -90.000,B 90.000,C 0.000} C_DIS
LIN {X 3.548,Y -45.269,Z -235.165,A -90.000,B 90.000,C 0.000} C_DIS
LIN {X 3.616,Y -45.333,Z -235.583,A -90.000,B 90.000,C 0.000} C_DIS
LIN {X 3.715,Y -45.445,Z -236.342,A -90.000,B 90.000,C 0.000} C_DIS
LIN {X 3.780,Y -45.529,Z -236.919,A -90.000,B 90.000,C 0.000} C_DIS
LIN {X 3.840,Y -45.618,Z -237.540,A -90.000,B 90.000,C 0.000} C_DIS
LIN {X 3.868,Y -45.664,Z -237.865,A -90.000,B 90.000,C 0.000} C_DIS
LIN {X 3.921,Y -45.758,Z -238.533,A -90.000,B 90.000,C 0.000} C_DIS
LIN {X 3.966,Y -45.854,Z -239.220,A -90.000,B 90.000,C 0.000} C_DIS
LIN {X 3.985,Y -45.901,Z -239.566,A -90.000,B 90.000,C 0.000} C_DIS
LIN {X 4.002,Y -45.942,Z -239.913,A -90.000,B 90.000,C 0.000} C_DIS
LIN {X 4.017,Y -45.971,Z -240.259,A -90.000,B 90.000,C 0.000} C_DIS
LIN {X 4.038,Y -46.024,Z -240.943,A -90.000,B 90.000,C 0.000} C_DIS
LIN {X 4.046,Y -46.050,Z -241.279,A -90.000,B 90.000,C 0.000} C_DIS
LIN {X 4.049,Y -46.075,Z -241.608,A -90.000,B 90.000,C 0.000} C_DIS
LIN {X 4.049,Y -46.123,Z -242.241,A -90.000,B 90.000,C 0.000} C_DIS
LIN {X 4.033,Y -46.166,Z -242.834,A -90.000,B 90.000,C 0.000} C_DIS
LIN {X 4.021,Y -46.188,Z -243.112,A -90.000,B 90.000,C 0.000} C_DIS
LIN {X 4.002,Y -46.214,Z -243.375,A -90.000,B 90.000,C 0.000} C_DIS
LIN {X 3.966,Y -46.249,Z -243.739,A -90.000,B 90.000,C 0.000} C_DIS
LIN {X 3.920,Y -46.278,Z -244.064,A -90.000,B 90.000,C 0.000} C_DIS
LIN {X 3.865,Y -46.303,Z -244.345,A -90.000,B 90.000,C 0.000} C_DIS
LIN {X 3.821,Y -46.315,Z -244.506,A -90.000,B 90.000,C 0.000} C_DIS
LIN {X 3.798,Y -46.319,Z -244.577,A -90.000,B 90.000,C 0.000} C_DIS
LIN {X 3.748,Y -46.324,Z -244.703,A -90.000,B 90.000,C 0.000} C_DIS
LIN {X 3.734,Y -46.324,Z -244.730,A -90.000,B 90.000,C 0.000} C_DIS
LIN {X 3.691,Y -46.325,Z -244.803,A -90.000,B 90.000,C 0.000} C_DIS
LIN {X 3.645,Y -46.325,Z -244.860,A -90.000,B 90.000,C 0.000} C_DIS
LIN {X 3.613,Y -46.324,Z -244.890,A -90.000,B 90.000,C 0.000} C_DIS
LIN {X 3.562,Y -46.323,Z -244.924,A -90.000,B 90.000,C 0.000} C_DIS
LIN {X 3.507,Y -46.322,Z -244.939,A -90.000,B 90.000,C 0.000} C_DIS
LIN {X 3.469,Y -46.321,Z -244.940,A -90.000,B 90.000,C 0.000} C_DIS
LIN {X 3.408,Y -46.317,Z -244.927,A -90.000,B 90.000,C 0.000} C_DIS
LIN {X 3.366,Y -46.313,Z -244.908,A -90.000,B 90.000,C 0.000} C_DIS
LIN {X 3.322,Y -46.308,Z -244.882,A -90.000,B 90.000,C 0.000} C_DIS
LIN {X 3.255,Y -46.300,Z -244.825,A -90.000,B 90.000,C 0.000} C_DIS
LIN {X 3.181,Y -46.290,Z -244.749,A -90.000,B 90.000,C 0.000} C_DIS
LIN {X 3.130,Y -46.281,Z -244.689,A -90.000,B 90.000,C 0.000} C_DIS
LIN {X 3.077,Y -46.270,Z -244.620,A -90.000,B 90.000,C 0.000} C_DIS
LIN {X 3.024,Y -46.257,Z -244.542,A -90.000,B 90.000,C 0.000} C_DIS
LIN {X 2.912,Y -46.229,Z -244.356,A -90.000,B 90.000,C 0.000} C_DIS
LIN {X 2.792,Y -46.197,Z -244.132,A -90.000,B 90.000,C 0.000} C_DIS
LIN {X 2.666,Y -46.160,Z -243.868,A -90.000,B 90.000,C 0.000} C_DIS
LIN {X 2.600,Y -46.139,Z -243.720,A -90.000,B 90.000,C 0.000} C_DIS
LIN {X 2.534,Y -46.118,Z -243.561,A -90.000,B 90.000,C 0.000} C_DIS
LIN {X 2.294,Y -46.040,Z -242.990,A -90.000,B 90.000,C 0.000} C_DIS
LIN {X 2.240,Y -46.021,Z -242.853,A -90.000,B 90.000,C 0.000} C_DIS
LIN {X 2.057,Y -45.954,Z -242.340,A -90.000,B 90.000,C 0.000} C_DIS
LIN {X 2.032,Y -45.945,Z -242.266,A -90.000,B 90.000,C 0.000} C_DIS
LIN {X 1.983,Y -45.926,Z -242.106,A -90.000,B 90.000,C 0.000} C_DIS
LIN {X 1.927,Y -45.894,Z -241.925,A -90.000,B 90.000,C 0.000} C_DIS
LIN {X 1.839,Y -45.850,Z -241.640,A -90.000,B 90.000,C 0.000} C_DIS
LIN {X 1.704,Y -45.779,Z -241.176,A -90.000,B 90.000,C 0.000} C_DIS
LIN {X 1.649,Y -45.747,Z -240.963,A -90.000,B 90.000,C 0.000} C_DIS
LIN {X 1.552,Y -45.688,Z -240.562,A -90.000,B 90.000,C 0.000} C_DIS
LIN {X 1.441,Y -45.610,Z -240.022,A -90.000,B 90.000,C 0.000} C_DIS
LIN {X 1.363,Y -45.545,Z -239.556,A -90.000,B 90.000,C 0.000} C_DIS
LIN {X 1.247,Y -45.422,Z -238.655,A -90.000,B 90.000,C 0.000} C_DIS
LIN {X 1.187,Y -45.340,Z -238.047,A -90.000,B 90.000,C 0.000} C_DIS
LIN {X 1.170,Y -45.308,Z -237.806,A -90.000,B 90.000,C 0.000} C_DIS
LIN {X 1.112,Y -45.195,Z -236.979,A -90.000,B 90.000,C 0.000} C_DIS
LIN {X 1.095,Y -45.148,Z -236.669,A -90.000,B 90.000,C 0.000} C_DIS
LIN {X 1.094,Y -45.139,Z -236.619,A -90.000,B 90.000,C 0.000} C_DIS
LIN {X 1.095,Y -45.131,Z -236.591,A -90.000,B 90.000,C 0.000} C_DIS
LIN {X 1.100,Y -45.129,Z -236.616,A -90.000,B 90.000,C 0.000} C_DIS
LIN {X 1.106,Y -45.132,Z -236.661,A -90.000,B 90.000,C 0.000} C_DIS
LIN {X 1.158,Y -45.244,Z -237.331,A -90.000,B 90.000,C 0.000} C_DIS
LIN {X 1.184,Y -45.296,Z -237.684,A -90.000,B 90.000,C 0.000} C_DIS
LIN {X 1.239,Y -45.407,Z -238.532,A -90.000,B 90.000,C 0.000} C_DIS
LIN {X 1.266,Y -45.469,Z -239.011,A -90.000,B 90.000,C 0.000} C_DIS
LIN {X 1.291,Y -45.534,Z -239.516,A -90.000,B 90.000,C 0.000} C_DIS
LIN {X 1.326,Y -45.634,Z -240.304,A -90.000,B 90.000,C 0.000} C_DIS
LIN {X 1.356,Y -45.769,Z -241.367,A -90.000,B 90.000,C 0.000} C_DIS
LIN {X 1.361,Y -45.804,Z -241.628,A -90.000,B 90.000,C 0.000} C_DIS
LIN {X 1.363,Y -45.884,Z -242.137,A -90.000,B 90.000,C 0.000} C_DIS
LIN {X 1.366,Y -45.915,Z -242.384,A -90.000,B 90.000,C 0.000} C_DIS
LIN {X 1.360,Y -45.955,Z -242.854,A -90.000,B 90.000,C 0.000} C_DIS
LIN {X 1.341,Y -45.996,Z -243.288,A -90.000,B 90.000,C 0.000} C_DIS
LIN {X 1.315,Y -46.034,Z -243.677,A -90.000,B 90.000,C 0.000} C_DIS
LIN {X 1.297,Y -46.050,Z -243.852,A -90.000,B 90.000,C 0.000} C_DIS
LIN {X 1.277,Y -46.065,Z -244.013,A -90.000,B 90.000,C 0.000} C_DIS
LIN {X 1.240,Y -46.084,Z -244.225,A -90.000,B 90.000,C 0.000} C_DIS
LIN {X 1.199,Y -46.099,Z -244.398,A -90.000,B 90.000,C 0.000} C_DIS
LIN {X 1.182,Y -46.103,Z -244.447,A -90.000,B 90.000,C 0.000} C_DIS
LIN {X 1.148,Y -46.109,Z -244.530,A -90.000,B 90.000,C 0.000} C_DIS
LIN {X 1.110,Y -46.112,Z -244.593,A -90.000,B 90.000,C 0.000} C_DIS
LIN {X 1.079,Y -46.113,Z -244.627,A -90.000,B 90.000,C 0.000} C_DIS
LIN {X 1.046,Y -46.113,Z -244.648,A -90.000,B 90.000,C 0.000} C_DIS
LIN {X 1.024,Y -46.112,Z -244.656,A -90.000,B 90.000,C 0.000} C_DIS
LIN {X 0.989,Y -46.109,Z -244.656,A -90.000,B 90.000,C 0.000} C_DIS
LIN {X 0.952,Y -46.105,Z -244.646,A -90.000,B 90.000,C 0.000} C_DIS
LIN {X 0.924,Y -46.101,Z -244.630,A -90.000,B 90.000,C 0.000} C_DIS
LIN {X 0.895,Y -46.097,Z -244.607,A -90.000,B 90.000,C 0.000} C_DIS
LIN {X 0.865,Y -46.091,Z -244.578,A -90.000,B 90.000,C 0.000} C_DIS
LIN {X 0.834,Y -46.085,Z -244.543,A -90.000,B 90.000,C 0.000} C_DIS
LIN {X 0.767,Y -46.071,Z -244.452,A -90.000,B 90.000,C 0.000} C_DIS
LIN {X 0.697,Y -46.053,Z -244.337,A -90.000,B 90.000,C 0.000} C_DIS
LIN {X 0.622,Y -46.032,Z -244.189,A -90.000,B 90.000,C 0.000} C_DIS
LIN {X 0.583,Y -46.020,Z -244.104,A -90.000,B 90.000,C 0.000} C_DIS
LIN {X 0.502,Y -45.994,Z -243.911,A -90.000,B 90.000,C 0.000} C_DIS
LIN {X 0.415,Y -45.970,Z -243.686,A -90.000,B 90.000,C 0.000} C_DIS
LIN {X 0.371,Y -45.954,Z -243.561,A -90.000,B 90.000,C 0.000} C_DIS
LIN {X 0.176,Y -45.897,Z -243.018,A -90.000,B 90.000,C 0.000} C_DIS
LIN {X 0.100,Y -45.873,Z -242.785,A -90.000,B 90.000,C 0.000} C_DIS
LIN {X -0.083,Y -45.765,Z -242.187,A -90.000,B 90.000,C 0.000} C_DIS
LIN {X -0.211,Y -45.685,Z -241.745,A -90.000,B 90.000,C 0.000} C_DIS
LIN {X -0.280,Y -45.637,Z -241.481,A -90.000,B 90.000,C 0.000} C_DIS
LIN {X -0.386,Y -45.559,Z -241.040,A -90.000,B 90.000,C 0.000} C_DIS
LIN {X -0.440,Y -45.514,Z -240.779,A -90.000,B 90.000,C 0.000} C_DIS
LIN {X -0.509,Y -45.465,Z -240.442,A -90.000,B 90.000,C 0.000} C_DIS
LIN {X -0.600,Y -45.390,Z -239.907,A -90.000,B 90.000,C 0.000} C_DIS
LIN {X -0.614,Y -45.376,Z -239.808,A -90.000,B 90.000,C 0.000} C_DIS
LIN {X -0.669,Y -45.308,Z -239.375,A -90.000,B 90.000,C 0.000} C_DIS
LIN {X -0.695,Y -45.282,Z -239.187,A -90.000,B 90.000,C 0.000} C_DIS
LIN {X -0.737,Y -45.229,Z -238.882,A -90.000,B 90.000,C 0.000} C_DIS
LIN {X -0.774,Y -45.191,Z -238.667,A -90.000,B 90.000,C 0.000} C_DIS
LIN {X -0.804,Y -45.165,Z -238.535,A -90.000,B 90.000,C 0.000} C_DIS
LIN {X -0.824,Y -45.155,Z -238.488,A -90.000,B 90.000,C 0.000} C_DIS
LIN {X -0.835,Y -45.152,Z -238.479,A -90.000,B 90.000,C 0.000} C_DIS
LIN {X -0.841,Y -45.151,Z -238.480,A -90.000,B 90.000,C 0.000} C_DIS
LIN {X -0.850,Y -45.153,Z -238.497,A -90.000,B 90.000,C 0.000} C_DIS
LIN {X -0.866,Y -45.163,Z -238.578,A -90.000,B 90.000,C 0.000} C_DIS
LIN {X -0.880,Y -45.183,Z -238.718,A -90.000,B 90.000,C 0.000} C_DIS
LIN {X -0.893,Y -45.229,Z -239.024,A -90.000,B 90.000,C 0.000} C_DIS
LIN {X -0.904,Y -45.315,Z -239.582,A -90.000,B 90.000,C 0.000} C_DIS
LIN {X -0.904,Y -45.361,Z -239.910,A -90.000,B 90.000,C 0.000} C_DIS
LIN {X -0.906,Y -45.404,Z -240.263,A -90.000,B 90.000,C 0.000} C_DIS
LIN {X -0.907,Y -45.456,Z -240.636,A -90.000,B 90.000,C 0.000} C_DIS
LIN {X -0.927,Y -45.638,Z -241.804,A -90.000,B 90.000,C 0.000} C_DIS
LIN {X -0.946,Y -45.726,Z -242.379,A -90.000,B 90.000,C 0.000} C_DIS
LIN {X -0.983,Y -45.833,Z -243.090,A -90.000,B 90.000,C 0.000} C_DIS
LIN {X -0.994,Y -45.850,Z -243.253,A -90.000,B 90.000,C 0.000} C_DIS
LIN {X -1.021,Y -45.875,Z -243.555,A -90.000,B 90.000,C 0.000} C_DIS
LIN {X -1.054,Y -45.895,Z -243.821,A -90.000,B 90.000,C 0.000} C_DIS
LIN {X -1.085,Y -45.908,Z -243.992,A -90.000,B 90.000,C 0.000} C_DIS
LIN {X -1.120,Y -45.918,Z -244.137,A -90.000,B 90.000,C 0.000} C_DIS
LIN {X -1.144,Y -45.923,Z -244.218,A -90.000,B 90.000,C 0.000} C_DIS
LIN {X -1.157,Y -45.925,Z -244.253,A -90.000,B 90.000,C 0.000} C_DIS
LIN {X -1.186,Y -45.929,Z -244.312,A -90.000,B 90.000,C 0.000} C_DIS
LIN {X -1.201,Y -45.930,Z -244.337,A -90.000,B 90.000,C 0.000} C_DIS
LIN {X -1.233,Y -45.931,Z -244.373,A -90.000,B 90.000,C 0.000} C_DIS
LIN {X -1.249,Y -45.931,Z -244.386,A -90.000,B 90.000,C 0.000} C_DIS
LIN {X -1.274,Y -45.931,Z -244.398,A -90.000,B 90.000,C 0.000} C_DIS
LIN {X -1.292,Y -45.930,Z -244.400,A -90.000,B 90.000,C 0.000} C_DIS
LIN {X -1.310,Y -45.929,Z -244.397,A -90.000,B 90.000,C 0.000} C_DIS
LIN {X -1.338,Y -45.926,Z -244.388,A -90.000,B 90.000,C 0.000} C_DIS
LIN {X -1.381,Y -45.921,Z -244.354,A -90.000,B 90.000,C 0.000} C_DIS
LIN {X -1.403,Y -45.918,Z -244.334,A -90.000,B 90.000,C 0.000} C_DIS
LIN {X -1.426,Y -45.914,Z -244.306,A -90.000,B 90.000,C 0.000} C_DIS
LIN {X -1.473,Y -45.906,Z -244.237,A -90.000,B 90.000,C 0.000} C_DIS
LIN {X -1.523,Y -45.895,Z -244.147,A -90.000,B 90.000,C 0.000} C_DIS
LIN {X -1.603,Y -45.875,Z -243.970,A -90.000,B 90.000,C 0.000} C_DIS
LIN {X -1.689,Y -45.851,Z -243.743,A -90.000,B 90.000,C 0.000} C_DIS
LIN {X -1.749,Y -45.830,Z -243.561,A -90.000,B 90.000,C 0.000} C_DIS
LIN {X -1.784,Y -45.819,Z -243.455,A -90.000,B 90.000,C 0.000} C_DIS
LIN {X -1.991,Y -45.697,Z -242.785,A -90.000,B 90.000,C 0.000} C_DIS
LIN {X -2.147,Y -45.598,Z -242.238,A -90.000,B 90.000,C 0.000} C_DIS
LIN {X -2.209,Y -45.555,Z -242.001,A -90.000,B 90.000,C 0.000} C_DIS
LIN {X -2.313,Y -45.479,Z -241.570,A -90.000,B 90.000,C 0.000} C_DIS
LIN {X -2.325,Y -45.473,Z -241.522,A -90.000,B 90.000,C 0.000} C_DIS
LIN {X -2.468,Y -45.390,Z -240.838,A -90.000,B 90.000,C 0.000} C_DIS
LIN {X -2.542,Y -45.308,Z -240.401,A -90.000,B 90.000,C 0.000} C_DIS
LIN {X -2.568,Y -45.285,Z -240.254,A -90.000,B 90.000,C 0.000} C_DIS
LIN {X -2.592,Y -45.260,Z -240.126,A -90.000,B 90.000,C 0.000} C_DIS
LIN {X -2.616,Y -45.238,Z -240.015,A -90.000,B 90.000,C 0.000} C_DIS
LIN {X -2.660,Y -45.204,Z -239.846,A -90.000,B 90.000,C 0.000} C_DIS
LIN {X -2.680,Y -45.191,Z -239.786,A -90.000,B 90.000,C 0.000} C_DIS
LIN {X -2.709,Y -45.178,Z -239.725,A -90.000,B 90.000,C 0.000} C_DIS
LIN {X -2.728,Y -45.173,Z -239.703,A -90.000,B 90.000,C 0.000} C_DIS
LIN {X -2.737,Y -45.171,Z -239.697,A -90.000,B 90.000,C 0.000} C_DIS
LIN {X -2.754,Y -45.170,Z -239.696,A -90.000,B 90.000,C 0.000} C_DIS
LIN {X -2.770,Y -45.171,Z -239.708,A -90.000,B 90.000,C 0.000} C_DIS
LIN {X -2.793,Y -45.177,Z -239.749,A -90.000,B 90.000,C 0.000} C_DIS
LIN {X -2.815,Y -45.188,Z -239.816,A -90.000,B 90.000,C 0.000} C_DIS
LIN {X -2.829,Y -45.198,Z -239.875,A -90.000,B 90.000,C 0.000} C_DIS
LIN {X -2.856,Y -45.223,Z -240.022,A -90.000,B 90.000,C 0.000} C_DIS
LIN {X -2.893,Y -45.274,Z -240.309,A -90.000,B 90.000,C 0.000} C_DIS
LIN {X -2.938,Y -45.359,Z -240.789,A -90.000,B 90.000,C 0.000} C_DIS
LIN {X -2.961,Y -45.396,Z -241.061,A -90.000,B 90.000,C 0.000} C_DIS
LIN {X -3.055,Y -45.527,Z -242.246,A -90.000,B 90.000,C 0.000} C_DIS
LIN {X -3.082,Y -45.571,Z -242.543,A -90.000,B 90.000,C 0.000} C_DIS
LIN {X -3.126,Y -45.634,Z -242.969,A -90.000,B 90.000,C 0.000} C_DIS
LIN {X -3.158,Y -45.673,Z -243.234,A -90.000,B 90.000,C 0.000} C_DIS
LIN {X -3.194,Y -45.708,Z -243.478,A -90.000,B 90.000,C 0.000} C_DIS
LIN {X -3.233,Y -45.739,Z -243.696,A -90.000,B 90.000,C 0.000} C_DIS
LIN {X -3.275,Y -45.763,Z -243.883,A -90.000,B 90.000,C 0.000} C_DIS
LIN {X -3.298,Y -45.772,Z -243.964,A -90.000,B 90.000,C 0.000} C_DIS
LIN {X -3.322,Y -45.778,Z -244.035,A -90.000,B 90.000,C 0.000} C_DIS
LIN {X -3.347,Y -45.785,Z -244.096,A -90.000,B 90.000,C 0.000} C_DIS
LIN {X -3.373,Y -45.791,Z -244.146,A -90.000,B 90.000,C 0.000} C_DIS
LIN {X -3.401,Y -45.795,Z -244.185,A -90.000,B 90.000,C 0.000} C_DIS
LIN {X -3.415,Y -45.796,Z -244.200,A -90.000,B 90.000,C 0.000} C_DIS
LIN {X -3.444,Y -45.797,Z -244.222,A -90.000,B 90.000,C 0.000} C_DIS
LIN {X -3.475,Y -45.796,Z -244.230,A -90.000,B 90.000,C 0.000} C_DIS
LIN {X -3.507,Y -45.793,Z -244.225,A -90.000,B 90.000,C 0.000} C_DIS
LIN {X -3.524,Y -45.791,Z -244.218,A -90.000,B 90.000,C 0.000} C_DIS
LIN {X -3.558,Y -45.784,Z -244.192,A -90.000,B 90.000,C 0.000} C_DIS
LIN {X -3.594,Y -45.774,Z -244.151,A -90.000,B 90.000,C 0.000} C_DIS
LIN {X -3.650,Y -45.758,Z -244.060,A -90.000,B 90.000,C 0.000} C_DIS
LIN {X -3.711,Y -45.736,Z -243.933,A -90.000,B 90.000,C 0.000} C_DIS
LIN {X -3.753,Y -45.715,Z -243.827,A -90.000,B 90.000,C 0.000} C_DIS
LIN {X -3.820,Y -45.680,Z -243.635,A -90.000,B 90.000,C 0.000} C_DIS
LIN {X -3.843,Y -45.661,Z -243.561,A -90.000,B 90.000,C 0.000} C_DIS
LIN {X -3.897,Y -45.629,Z -243.385,A -90.000,B 90.000,C 0.000} C_DIS
LIN {X -3.944,Y -45.600,Z -243.221,A -90.000,B 90.000,C 0.000} C_DIS
LIN {X -4.052,Y -45.553,Z -242.848,A -90.000,B 90.000,C 0.000} C_DIS
LIN {X -4.132,Y -45.516,Z -242.552,A -90.000,B 90.000,C 0.000} C_DIS
LIN {X -4.267,Y -45.449,Z -241.999,A -90.000,B 90.000,C 0.000} C_DIS
LIN {X -4.371,Y -45.389,Z -241.506,A -90.000,B 90.000,C 0.000} C_DIS
LIN {X -4.422,Y -45.342,Z -241.261,A -90.000,B 90.000,C 0.000} C_DIS
LIN {X -4.453,Y -45.308,Z -241.085,A -90.000,B 90.000,C 0.000} C_DIS
LIN {X -4.453,Y -60.000,Z -241.085,A -90.000,B 90.000,C 0.000} C_DIS
LIN {X -58.261,Y -60.000,Z -243.561,A -90.000,B 90.000,C 0.000} C_DIS
LIN {X -58.261,Y -46.933,Z -243.561,A -90.000,B 90.000,C 0.000} C_DIS
LIN {X -58.247,Y -46.883,Z -243.441,A -90.000,B 90.000,C 0.000} C_DIS
LIN {X -58.236,Y -46.857,Z -243.378,A -90.000,B 90.000,C 0.000} C_DIS
LIN {X -58.203,Y -46.800,Z -243.234,A -90.000,B 90.000,C 0.000} C_DIS
LIN {X -58.163,Y -46.752,Z -243.107,A -90.000,B 90.000,C 0.000} C_DIS
LIN {X -58.116,Y -46.709,Z -242.988,A -90.000,B 90.000,C 0.000} C_DIS
LIN {X -58.031,Y -46.649,Z -242.815,A -90.000,B 90.000,C 0.000} C_DIS
LIN {X -57.987,Y -46.625,Z -242.740,A -90.000,B 90.000,C 0.000} C_DIS
LIN {X -57.956,Y -46.610,Z -242.692,A -90.000,B 90.000,C 0.000} C_DIS
LIN {X -57.895,Y -46.583,Z -242.603,A -90.000,B 90.000,C 0.000} C_DIS
LIN {X -57.548,Y -46.490,Z -242.233,A -90.000,B 90.000,C 0.000} C_DIS
LIN {X -57.016,Y -46.449,Z -241.905,A -90.000,B 90.000,C 0.000} C_DIS
LIN {X -56.113,Y -46.450,Z -241.513,A -90.000,B 90.000,C 0.000} C_DIS
LIN {X -54.342,Y -46.474,Z -240.796,A -90.000,B 90.000,C 0.000} C_DIS
LIN {X -54.254,Y -46.476,Z -240.762,A -90.000,B 90.000,C 0.000} C_DIS
LIN {X -52.709,Y -46.531,Z -240.215,A -90.000,B 90.000,C 0.000} C_DIS
LIN {X -51.217,Y -46.570,Z -239.695,A -90.000,B 90.000,C 0.000} C_DIS
LIN {X -49.890,Y -46.612,Z -239.275,A -90.000,B 90.000,C 0.000} C_DIS
LIN {X -48.664,Y -46.631,Z -238.894,A -90.000,B 90.000,C 0.000} C_DIS
LIN {X -47.676,Y -46.632,Z -238.595,A -90.000,B 90.000,C 0.000} C_DIS
LIN {X -45.875,Y -46.646,Z -238.089,A -90.000,B 90.000,C 0.000} C_DIS
LIN {X -45.004,Y -46.648,Z -237.848,A -90.000,B 90.000,C 0.000} C_DIS
LIN {X -43.818,Y -46.673,Z -237.595,A -90.000,B 90.000,C 0.000} C_DIS
LIN {X -43.730,Y -46.676,Z -237.578,A -90.000,B 90.000,C 0.000} C_DIS
LIN {X -42.503,Y -46.722,Z -237.372,A -90.000,B 90.000,C 0.000} C_DIS
LIN {X -42.428,Y -46.725,Z -237.361,A -90.000,B 90.000,C 0.000} C_DIS
LIN {X -41.513,Y -46.770,Z -237.242,A -90.000,B 90.000,C 0.000} C_DIS
LIN {X -41.101,Y -46.786,Z -237.190,A -90.000,B 90.000,C 0.000} C_DIS
LIN {X -40.131,Y -46.804,Z -237.073,A -90.000,B 90.000,C 0.000} C_DIS
LIN {X -38.373,Y -46.804,Z -236.873,A -90.000,B 90.000,C 0.000} C_DIS
LIN {X -37.605,Y -46.812,Z -236.816,A -90.000,B 90.000,C 0.000} C_DIS
LIN {X -37.486,Y -46.814,Z -236.810,A -90.000,B 90.000,C 0.000} C_DIS
LIN {X -37.249,Y -46.820,Z -236.806,A -90.000,B 90.000,C 0.000} C_DIS
LIN {X -37.004,Y -46.830,Z -236.817,A -90.000,B 90.000,C 0.000} C_DIS
LIN {X -35.134,Y -46.919,Z -237.034,A -90.000,B 90.000,C 0.000} C_DIS
LIN {X -34.934,Y -46.925,Z -237.059,A -90.000,B 90.000,C 0.000} C_DIS
LIN {X -34.210,Y -46.925,Z -237.151,A -90.000,B 90.000,C 0.000} C_DIS
LIN {X -34.101,Y -46.925,Z -237.168,A -90.000,B 90.000,C 0.000} C_DIS
LIN {X -33.424,Y -46.933,Z -237.296,A -90.000,B 90.000,C 0.000} C_DIS
LIN {X -32.159,Y -46.934,Z -237.543,A -90.000,B 90.000,C 0.000} C_DIS
LIN {X -31.990,Y -46.937,Z -237.590,A -90.000,B 90.000,C 0.000} C_DIS
LIN {X -31.819,Y -46.941,Z -237.646,A -90.000,B 90.000,C 0.000} C_DIS
LIN {X -31.562,Y -46.951,Z -237.749,A -90.000,B 90.000,C 0.000} C_DIS
LIN {X -30.821,Y -46.991,Z -238.108,A -90.000,B 90.000,C 0.000} C_DIS
LIN {X -30.683,Y -46.995,Z -238.175,A -90.000,B 90.000,C 0.000} C_DIS
LIN {X -30.137,Y -46.995,Z -238.446,A -90.000,B 90.000,C 0.000} C_DIS
LIN {X -30.068,Y -46.995,Z -238.482,A -90.000,B 90.000,C 0.000} C_DIS
LIN {X -29.972,Y -46.995,Z -238.537,A -90.000,B 90.000,C 0.000} C_DIS
LIN {X -28.530,Y -46.995,Z -239.427,A -90.000,B 90.000,C 0.000} C_DIS
LIN {X -28.367,Y -46.996,Z -239.538,A -90.000,B 90.000,C 0.000} C_DIS
LIN {X -28.086,Y -47.004,Z -239.768,A -90.000,B 90.000,C 0.000} C_DIS
LIN {X -27.908,Y -47.013,Z -239.952,A -90.000,B 90.000,C 0.000} C_DIS
LIN {X -27.443,Y -47.013,Z -240.440,A -90.000,B 90.000,C 0.000} C_DIS
LIN {X -26.934,Y -47.003,Z -240.979,A -90.000,B 90.000,C 0.000} C_DIS
LIN {X -26.778,Y -47.001,Z -241.165,A -90.000,B 90.000,C 0.000} C_DIS
LIN {X -25.854,Y -47.001,Z -242.345,A -90.000,B 90.000,C 0.000} C_DIS
LIN {X -25.551,Y -47.007,Z -242.892,A -90.000,B 90.000,C 0.000} C_DIS
LIN {X -25.430,Y -47.043,Z -243.505,A -90.000,B 90.000,C 0.000} C_DIS
LIN {X -25.429,Y -47.048,Z -243.561,A -90.000,B 90.000,C 0.000} C_DIS
LIN {X -25.429,Y -60.000,Z -243.561,A -90.000,B 90.000,C 0.000} C_DIS
LIN {X -60.226,Y -60.000,Z -243.561,A -90.000,B 90.000,C 0.000} C_DIS
LIN {X -60.226,Y -46.558,Z -243.561,A -90.000,B 90.000,C 0.000} C_DIS
LIN {X -60.199,Y -46.462,Z -243.327,A -90.000,B 90.000,C 0.000} C_DIS
LIN {X -60.174,Y -46.404,Z -243.181,A -90.000,B 90.000,C 0.000} C_DIS
LIN {X -60.114,Y -46.302,Z -242.917,A -90.000,B 90.000,C 0.000} C_DIS
LIN {X -60.051,Y -46.219,Z -242.717,A -90.000,B 90.000,C 0.000} C_DIS
LIN {X -60.000,Y -46.164,Z -242.578,A -90.000,B 90.000,C 0.000} C_DIS
LIN {X -59.958,Y -46.122,Z -242.474,A -90.000,B 90.000,C 0.000} C_DIS
LIN {X -59.910,Y -46.081,Z -242.366,A -90.000,B 90.000,C 0.000} C_DIS
LIN {X -59.792,Y -45.992,Z -242.131,A -90.000,B 90.000,C 0.000} C_DIS
LIN {X -59.707,Y -45.938,Z -241.984,A -90.000,B 90.000,C 0.000} C_DIS
LIN {X -59.627,Y -45.892,Z -241.857,A -90.000,B 90.000,C 0.000} C_DIS
LIN {X -59.520,Y -45.840,Z -241.704,A -90.000,B 90.000,C 0.000} C_DIS
LIN {X -59.374,Y -45.782,Z -241.521,A -90.000,B 90.000,C 0.000} C_DIS
LIN {X -58.975,Y -45.665,Z -241.100,A -90.000,B 90.000,C 0.000} C_DIS
LIN {X -58.853,Y -45.635,Z -240.982,A -90.000,B 90.000,C 0.000} C_DIS
LIN {X -58.536,Y -45.591,Z -240.744,A -90.000,B 90.000,C 0.000} C_DIS
LIN {X -57.968,Y -45.551,Z -240.392,A -90.000,B 90.000,C 0.000} C_DIS
LIN {X -57.727,Y -45.547,Z -240.267,A -90.000,B 90.000,C 0.000} C_DIS
LIN {X -56.827,Y -45.565,Z -239.867,A -90.000,B 90.000,C 0.000} C_DIS
LIN {X -56.219,Y -45.586,Z -239.613,A -90.000,B 90.000,C 0.000} C_DIS
LIN {X -55.011,Y -45.621,Z -239.115,A -90.000,B 90.000,C 0.000} C_DIS
LIN {X -54.877,Y -45.626,Z -239.063,A -90.000,B 90.000,C 0.000} C_DIS
LIN {X -54.659,Y -45.635,Z -238.984,A -90.000,B 90.000,C 0.000} C_DIS
LIN {X -51.791,Y -45.711,Z -237.982,A -90.000,B 90.000,C 0.000} C_DIS
LIN {X -49.716,Y -45.791,Z -237.316,A -90.000,B 90.000,C 0.000} C_DIS
LIN {X -48.207,Y -45.838,Z -236.838,A -90.000,B 90.000,C 0.000} C_DIS
LIN {X -45.503,Y -45.947,Z -236.042,A -90.000,B 90.000,C 0.000} C_DIS
LIN {X -45.381,Y -45.954,Z -236.010,A -90.000,B 90.000,C 0.000} C_DIS
LIN {X -45.236,Y -45.964,Z -235.977,A -90.000,B 90.000,C 0.000} C_DIS
LIN {X -44.742,Y -45.989,Z -235.866,A -90.000,B 90.000,C 0.000} C_DIS
LIN {X -44.290,Y -46.008,Z -235.767,A -90.000,B 90.000,C 0.000} C_DIS
LIN {X -44.064,Y -46.017,Z -235.720,A -90.000,B 90.000,C 0.000} C_DIS
LIN {X -42.792,Y -46.063,Z -235.506,A -90.000,B 90.000,C 0.000} C_DIS
LIN {X -42.679,Y -46.068,Z -235.489,A -90.000,B 90.000,C 0.000} C_DIS
LIN {X -40.135,Y -46.192,Z -235.157,A -90.000,B 90.000,C 0.000} C_DIS
LIN {X -38.523,Y -46.256,Z -234.956,A -90.000,B 90.000,C 0.000} C_DIS
LIN {X -37.907,Y -46.288,Z -234.902,A -90.000,B 90.000,C 0.000} C_DIS
LIN {X -37.744,Y -46.293,Z -234.889,A -90.000,B 90.000,C 0.000} C_DIS
LIN {X -37.563,Y -46.300,Z -234.879,A -90.000,B 90.000,C 0.000} C_DIS
LIN {X -37.269,Y -46.313,Z -234.872,A -90.000,B 90.000,C 0.000} C_DIS
LIN {X -37.147,Y -46.320,Z -234.872,A -90.000,B 90.000,C 0.000} C_DIS
LIN {X -37.063,Y -46.325,Z -234.875,A -90.000,B 90.000,C 0.000} C_DIS
LIN {X -36.902,Y -46.332,Z -234.882,A -90.000,B 90.000,C 0.000} C_DIS
LIN {X -36.757,Y -46.339,Z -234.894,A -90.000,B 90.000,C 0.000} C_DIS
LIN {X -36.013,Y -46.383,Z -234.978,A -90.000,B 90.000,C 0.000} C_DIS
LIN {X -34.550,Y -46.453,Z -235.148,A -90.000,B 90.000,C 0.000} C_DIS
LIN {X -33.964,Y -46.481,Z -235.216,A -90.000,B 90.000,C 0.000} C_DIS
LIN {X -33.800,Y -46.490,Z -235.239,A -90.000,B 90.000,C 0.000} C_DIS
LIN {X -32.908,Y -46.546,Z -235.398,A -90.000,B 90.000,C 0.000} C_DIS
LIN {X -32.721,Y -46.555,Z -235.432,A -90.000,B 90.000,C 0.000} C_DIS
LIN {X -32.490,Y -46.558,Z -235.477,A -90.000,B 90.000,C 0.000} C_DIS
LIN {X -31.855,Y -46.559,Z -235.601,A -90.000,B 90.000,C 0.000} C_DIS
LIN {X -31.679,Y -46.560,Z -235.638,A -90.000,B 90.000,C 0.000} C_DIS
LIN {X -31.486,Y -46.564,Z -235.691,A -90.000,B 90.000,C 0.000} C_DIS
LIN {X -31.375,Y -46.566,Z -235.724,A -90.000,B 90.000,C 0.000} C_DIS
LIN {X -31.204,Y -46.571,Z -235.779,A -90.000,B 90.000,C 0.000} C_DIS
LIN {X -31.074,Y -46.575,Z -235.826,A -90.000,B 90.000,C 0.000} C_DIS
LIN {X -30.816,Y -46.585,Z -235.930,A -90.000,B 90.000,C 0.000} C_DIS
LIN {X -30.688,Y -46.591,Z -235.986,A -90.000,B 90.000,C 0.000} C_DIS
LIN {X -29.227,Y -46.672,Z -236.694,A -90.000,B 90.000,C 0.000} C_DIS
LIN {X -29.069,Y -46.680,Z -236.778,A -90.000,B 90.000,C 0.000} C_DIS
LIN {X -28.940,Y -46.685,Z -236.852,A -90.000,B 90.000,C 0.000} C_DIS
LIN {X -27.492,Y -46.686,Z -237.746,A -90.000,B 90.000,C 0.000} C_DIS
LIN {X -27.257,Y -46.688,Z -237.903,A -90.000,B 90.000,C 0.000} C_DIS
LIN {X -27.136,Y -46.690,Z -237.992,A -90.000,B 90.000,C 0.000} C_DIS
LIN {X -26.830,Y -46.698,Z -238.242,A -90.000,B 90.000,C 0.000} C_DIS
LIN {X -26.658,Y -46.704,Z -238.400,A -90.000,B 90.000,C 0.000} C_DIS
LIN {X -26.341,Y -46.718,Z -238.728,A -90.000,B 90.000,C 0.000} C_DIS
LIN {X -25.500,Y -46.699,Z -239.618,A -90.000,B 90.000,C 0.000} C_DIS
LIN {X -25.422,Y -46.698,Z -239.705,A -90.000,B 90.000,C 0.000} C_DIS
LIN {X -25.221,Y -46.696,Z -239.947,A -90.000,B 90.000,C 0.000} C_DIS
LIN {X -24.328,Y -46.694,Z -241.088,A -90.000,B 90.000,C 0.000} C_DIS
LIN {X -24.242,Y -46.692,Z -241.202,A -90.000,B 90.000,C 0.000} C_DIS
LIN {X -24.177,Y -46.691,Z -241.301,A -90.000,B 90.000,C 0.000} C_DIS
LIN {X -24.124,Y -46.691,Z -241.390,A -90.000,B 90.000,C 0.000} C_DIS
LIN {X -23.822,Y -46.692,Z -241.938,A -90.000,B 90.000,C 0.000} C_DIS
LIN {X -23.608,Y -46.709,Z -242.525,A -90.000,B 90.000,C 0.000} C_DIS
LIN {X -23.487,Y -46.741,Z -243.138,A -90.000,B 90.000,C 0.000} C_DIS
LIN {X -23.450,Y -46.763,Z -243.478,A -90.000,B 90.000,C 0.000} C_DIS
LIN {X -23.448,Y -46.770,Z -243.561,A -90.000,B 90.000,C 0.000} C_DIS
LIN {X -23.448,Y -60.000,Z -243.561,A -90.000,B 90.000,C 0.000} C_DIS
LIN {X -43.239,Y -60.000,Z -233.701,A -90.000,B 90.000,C 0.000} C_DIS
LIN {X -43.239,Y -45.308,Z -233.701,A -90.000,B 90.000,C 0.000} C_DIS
LIN {X -42.929,Y -45.332,Z -233.646,A -90.000,B 90.000,C 0.000} C_DIS
LIN {X -41.646,Y -45.448,Z -233.457,A -90.000,B 90.000,C 0.000} C_DIS
LIN {X -40.697,Y -45.518,Z -233.325,A -90.000,B 90.000,C 0.000} C_DIS
LIN {X -38.819,Y -45.612,Z -233.083,A -90.000,B 90.000,C 0.000} C_DIS
LIN {X -38.661,Y -45.619,Z -233.065,A -90.000,B 90.000,C 0.000} C_DIS
LIN {X -37.877,Y -45.660,Z -232.997,A -90.000,B 90.000,C 0.000} C_DIS
LIN {X -37.646,Y -45.673,Z -232.981,A -90.000,B 90.000,C 0.000} C_DIS
LIN {X -37.282,Y -45.699,Z -232.968,A -90.000,B 90.000,C 0.000} C_DIS
LIN {X -37.100,Y -45.713,Z -232.967,A -90.000,B 90.000,C 0.000} C_DIS
LIN {X -36.724,Y -45.747,Z -232.978,A -90.000,B 90.000,C 0.000} C_DIS
LIN {X -36.508,Y -45.769,Z -232.993,A -90.000,B 90.000,C 0.000} C_DIS
LIN {X -35.408,Y -45.894,Z -233.101,A -90.000,B 90.000,C 0.000} C_DIS
LIN {X -34.713,Y -45.953,Z -233.175,A -90.000,B 90.000,C 0.000} C_DIS
LIN {X -33.718,Y -46.004,Z -233.290,A -90.000,B 90.000,C 0.000} C_DIS
LIN {X -33.460,Y -46.018,Z -233.325,A -90.000,B 90.000,C 0.000} C_DIS
LIN {X -32.910,Y -46.054,Z -233.422,A -90.000,B 90.000,C 0.000} C_DIS
LIN {X -31.543,Y -46.145,Z -233.668,A -90.000,B 90.000,C 0.000} C_DIS
LIN {X -31.278,Y -46.160,Z -233.720,A -90.000,B 90.000,C 0.000} C_DIS
LIN {X -31.166,Y -46.168,Z -233.745,A -90.000,B 90.000,C 0.000} C_DIS
LIN {X -30.839,Y -46.193,Z -233.833,A -90.000,B 90.000,C 0.000} C_DIS
LIN {X -30.681,Y -46.204,Z -233.881,A -90.000,B 90.000,C 0.000} C_DIS
LIN {X -30.589,Y -46.209,Z -233.910,A -90.000,B 90.000,C 0.000} C_DIS
LIN {X -30.392,Y -46.217,Z -233.980,A -90.000,B 90.000,C 0.000} C_DIS
LIN {X -30.070,Y -46.231,Z -234.108,A -90.000,B 90.000,C 0.000} C_DIS
LIN {X -29.878,Y -46.240,Z -234.192,A -90.000,B 90.000,C 0.000} C_DIS
LIN {X -29.476,Y -46.262,Z -234.385,A -90.000,B 90.000,C 0.000} C_DIS
LIN {X -28.353,Y -46.324,Z -234.929,A -90.000,B 90.000,C 0.000} C_DIS
LIN {X -28.139,Y -46.335,Z -235.041,A -90.000,B 90.000,C 0.000} C_DIS
LIN {X -27.942,Y -46.347,Z -235.152,A -90.000,B 90.000,C 0.000} C_DIS
LIN {X -27.385,Y -46.383,Z -235.489,A -90.000,B 90.000,C 0.000} C_DIS
LIN {X -27.266,Y -46.388,Z -235.561,A -90.000,B 90.000,C 0.000} C_DIS
LIN {X -26.453,Y -46.389,Z -236.063,A -90.000,B 90.000,C 0.000} C_DIS
LIN {X -26.157,Y -46.391,Z -236.259,A -90.000,B 90.000,C 0.000} C_DIS
LIN {X -26.014,Y -46.393,Z -236.361,A -90.000,B 90.000,C 0.000} C_DIS
LIN {X -25.880,Y -46.395,Z -236.463,A -90.000,B 90.000,C 0.000} C_DIS
LIN {X -25.545,Y -46.404,Z -236.738,A -90.000,B 90.000,C 0.000} C_DIS
LIN {X -25.349,Y -46.409,Z -236.916,A -90.000,B 90.000,C 0.000} C_DIS
LIN {X -25.228,Y -46.412,Z -237.033,A -90.000,B 90.000,C 0.000} C_DIS
LIN {X -24.783,Y -46.430,Z -237.495,A -90.000,B 90.000,C 0.000} C_DIS
LIN {X -24.078,Y -46.415,Z -238.241,A -90.000,B 90.000,C 0.000} C_DIS
LIN {X -24.005,Y -46.413,Z -238.320,A -90.000,B 90.000,C 0.000} C_DIS
LIN {X -23.876,Y -46.411,Z -238.470,A -90.000,B 90.000,C 0.000} C_DIS
LIN {X -23.702,Y -46.409,Z -238.678,A -90.000,B 90.000,C 0.000} C_DIS
LIN {X -23.254,Y -46.407,Z -239.250,A -90.000,B 90.000,C 0.000} C_DIS
LIN {X -22.794,Y -46.398,Z -239.838,A -90.000,B 90.000,C 0.000} C_DIS
LIN {X -22.699,Y -46.394,Z -239.964,A -90.000,B 90.000,C 0.000} C_DIS
LIN {X -22.596,Y -46.390,Z -240.107,A -90.000,B 90.000,C 0.000} C_DIS
LIN {X -22.530,Y -46.389,Z -240.207,A -90.000,B 90.000,C 0.000} C_DIS
LIN {X -22.471,Y -46.387,Z -240.301,A -90.000,B 90.000,C 0.000} C_DIS
LIN {X -22.432,Y -46.387,Z -240.368,A -90.000,B 90.000,C 0.000} C_DIS
LIN {X -22.092,Y -46.385,Z -240.983,A -90.000,B 90.000,C 0.000} C_DIS
LIN {X -21.962,Y -46.388,Z -241.268,A -90.000,B 90.000,C 0.000} C_DIS
LIN {X -21.748,Y -46.401,Z -241.856,A -90.000,B 90.000,C 0.000} C_DIS
LIN {X -21.706,Y -46.404,Z -241.986,A -90.000,B 90.000,C 0.000} C_DIS
LIN {X -21.664,Y -46.411,Z -242.159,A -90.000,B 90.000,C 0.000} C_DIS
LIN {X -21.568,Y -46.433,Z -242.653,A -90.000,B 90.000,C 0.000} C_DIS
LIN {X -21.537,Y -46.442,Z -242.814,A -90.000,B 90.000,C 0.000} C_DIS
LIN {X -21.518,Y -46.450,Z -242.941,A -90.000,B 90.000,C 0.000} C_DIS
LIN {X -21.481,Y -46.474,Z -243.280,A -90.000,B 90.000,C 0.000} C_DIS
LIN {X -21.469,Y -46.487,Z -243.455,A -90.000,B 90.000,C 0.000} C_DIS
LIN {X -21.467,Y -46.496,Z -243.561,A -90.000,B 90.000,C 0.000} C_DIS
LIN {X -21.467,Y -60.000,Z -243.561,A -90.000,B 90.000,C 0.000} C_DIS
LIN {X -35.058,Y -60.000,Z -231.218,A -90.000,B 90.000,C 0.000} C_DIS
LIN {X -35.058,Y -45.308,Z -231.218,A -90.000,B 90.000,C 0.000} C_DIS
LIN {X -34.097,Y -45.420,Z -231.311,A -90.000,B 90.000,C 0.000} C_DIS
LIN {X -33.424,Y -45.491,Z -231.379,A -90.000,B 90.000,C 0.000} C_DIS
LIN {X -33.092,Y -45.529,Z -231.421,A -90.000,B 90.000,C 0.000} C_DIS
LIN {X -32.536,Y -45.587,Z -231.514,A -90.000,B 90.000,C 0.000} C_DIS
LIN {X -32.416,Y -45.599,Z -231.535,A -90.000,B 90.000,C 0.000} C_DIS
LIN {X -31.189,Y -45.680,Z -231.755,A -90.000,B 90.000,C 0.000} C_DIS
LIN {X -30.841,Y -45.704,Z -231.822,A -90.000,B 90.000,C 0.000} C_DIS
LIN {X -30.629,Y -45.721,Z -231.871,A -90.000,B 90.000,C 0.000} C_DIS
LIN {X -30.239,Y -45.752,Z -231.977,A -90.000,B 90.000,C 0.000} C_DIS
LIN {X -29.981,Y -45.774,Z -232.055,A -90.000,B 90.000,C 0.000} C_DIS
LIN {X -29.724,Y -45.798,Z -232.142,A -90.000,B 90.000,C 0.000} C_DIS
LIN {X -29.294,Y -45.843,Z -232.306,A -90.000,B 90.000,C 0.000} C_DIS
LIN {X -29.009,Y -45.876,Z -232.428,A -90.000,B 90.000,C 0.000} C_DIS
LIN {X -28.799,Y -45.900,Z -232.526,A -90.000,B 90.000,C 0.000} C_DIS
LIN {X -28.445,Y -45.922,Z -232.696,A -90.000,B 90.000,C 0.000} C_DIS
LIN {X -27.478,Y -45.976,Z -233.165,A -90.000,B 90.000,C 0.000} C_DIS
LIN {X -27.226,Y -45.990,Z -233.295,A -90.000,B 90.000,C 0.000} C_DIS
LIN {X -26.956,Y -46.006,Z -233.446,A -90.000,B 90.000,C 0.000} C_DIS
LIN {X -25.727,Y -46.085,Z -234.188,A -90.000,B 90.000,C 0.000} C_DIS
LIN {X -25.569,Y -46.092,Z -234.285,A -90.000,B 90.000,C 0.000} C_DIS
LIN {X -25.415,Y -46.092,Z -234.380,A -90.000,B 90.000,C 0.000} C_DIS
LIN {X -25.064,Y -46.094,Z -234.611,A -90.000,B 90.000,C 0.000} C_DIS
LIN {X -24.893,Y -46.096,Z -234.732,A -90.000,B 90.000,C 0.000} C_DIS
LIN {X -24.678,Y -46.100,Z -234.892,A -90.000,B 90.000,C 0.000} C_DIS
LIN {X -24.444,Y -46.104,Z -235.083,A -90.000,B 90.000,C 0.000} C_DIS
LIN {X -24.359,Y -46.105,Z -235.152,A -90.000,B 90.000,C 0.000} C_DIS
LIN {X -24.218,Y -46.107,Z -235.271,A -90.000,B 90.000,C 0.000} C_DIS
LIN {X -23.985,Y -46.113,Z -235.484,A -90.000,B 90.000,C 0.000} C_DIS
LIN {X -23.796,Y -46.119,Z -235.667,A -90.000,B 90.000,C 0.000} C_DIS
LIN {X -23.225,Y -46.142,Z -236.262,A -90.000,B 90.000,C 0.000} C_DIS
LIN {X -22.718,Y -46.131,Z -236.797,A -90.000,B 90.000,C 0.000} C_DIS
LIN {X -22.545,Y -46.127,Z -236.984,A -90.000,B 90.000,C 0.000} C_DIS
LIN {X -22.382,Y -46.125,Z -237.171,A -90.000,B 90.000,C 0.000} C_DIS
LIN {X -22.185,Y -46.121,Z -237.406,A -90.000,B 90.000,C 0.000} C_DIS
LIN {X -21.320,Y -46.105,Z -238.512,A -90.000,B 90.000,C 0.000} C_DIS
LIN {X -21.129,Y -46.098,Z -238.761,A -90.000,B 90.000,C 0.000} C_DIS
LIN {X -21.010,Y -46.094,Z -238.925,A -90.000,B 90.000,C 0.000} C_DIS
LIN {X -20.883,Y -46.090,Z -239.112,A -90.000,B 90.000,C 0.000} C_DIS
LIN {X -20.794,Y -46.088,Z -239.253,A -90.000,B 90.000,C 0.000} C_DIS
LIN {X -20.722,Y -46.087,Z -239.375,A -90.000,B 90.000,C 0.000} C_DIS
LIN {X -20.334,Y -46.085,Z -240.077,A -90.000,B 90.000,C 0.000} C_DIS
LIN {X -20.272,Y -46.086,Z -240.209,A -90.000,B 90.000,C 0.000} C_DIS
LIN {X -20.160,Y -46.088,Z -240.453,A -90.000,B 90.000,C 0.000} C_DIS
LIN {X -20.108,Y -46.089,Z -240.580,A -90.000,B 90.000,C 0.000} C_DIS
LIN {X -19.891,Y -46.102,Z -241.179,A -90.000,B 90.000,C 0.000} C_DIS
LIN {X -19.823,Y -46.108,Z -241.381,A -90.000,B 90.000,C 0.000} C_DIS
LIN {X -19.780,Y -46.114,Z -241.532,A -90.000,B 90.000,C 0.000} C_DIS
LIN {X -19.722,Y -46.125,Z -241.778,A -90.000,B 90.000,C 0.000} C_DIS
LIN {X -19.583,Y -46.161,Z -242.487,A -90.000,B 90.000,C 0.000} C_DIS
LIN {X -19.546,Y -46.176,Z -242.749,A -90.000,B 90.000,C 0.000} C_DIS
LIN {X -19.510,Y -46.197,Z -243.082,A -90.000,B 90.000,C 0.000} C_DIS
LIN {X -19.502,Y -46.203,Z -243.169,A -90.000,B 90.000,C 0.000} C_DIS
LIN {X -19.491,Y -46.214,Z -243.344,A -90.000,B 90.000,C 0.000} C_DIS
LIN {X -19.485,Y -46.230,Z -243.561,A -90.000,B 90.000,C 0.000} C_DIS
LIN {X -19.485,Y -60.000,Z -243.561,A -90.000,B 90.000,C 0.000} C_DIS
LIN {X -29.656,Y -60.000,Z -230.116,A -90.000,B 90.000,C 0.000} C_DIS
LIN {X -29.656,Y -45.308,Z -230.116,A -90.000,B 90.000,C 0.000} C_DIS
LIN {X -29.377,Y -45.335,Z -230.200,A -90.000,B 90.000,C 0.000} C_DIS
LIN {X -29.063,Y -45.364,Z -230.305,A -90.000,B 90.000,C 0.000} C_DIS
LIN {X -28.550,Y -45.417,Z -230.499,A -90.000,B 90.000,C 0.000} C_DIS
LIN {X -28.202,Y -45.456,Z -230.647,A -90.000,B 90.000,C 0.000} C_DIS
LIN {X -27.252,Y -45.574,Z -231.090,A -90.000,B 90.000,C 0.000} C_DIS
LIN {X -27.021,Y -45.601,Z -231.199,A -90.000,B 90.000,C 0.000} C_DIS
LIN {X -26.623,Y -45.627,Z -231.391,A -90.000,B 90.000,C 0.000} C_DIS
LIN {X -26.305,Y -45.646,Z -231.553,A -90.000,B 90.000,C 0.000} C_DIS
LIN {X -25.980,Y -45.664,Z -231.735,A -90.000,B 90.000,C 0.000} C_DIS
LIN {X -24.378,Y -45.767,Z -232.701,A -90.000,B 90.000,C 0.000} C_DIS
LIN {X -24.033,Y -45.791,Z -232.923,A -90.000,B 90.000,C 0.000} C_DIS
LIN {X -23.907,Y -45.798,Z -233.007,A -90.000,B 90.000,C 0.000} C_DIS
LIN {X -23.772,Y -45.800,Z -233.102,A -90.000,B 90.000,C 0.000} C_DIS
LIN {X -23.491,Y -45.802,Z -233.311,A -90.000,B 90.000,C 0.000} C_DIS
LIN {X -23.187,Y -45.806,Z -233.556,A -90.000,B 90.000,C 0.000} C_DIS
LIN {X -22.943,Y -45.809,Z -233.759,A -90.000,B 90.000,C 0.000} C_DIS
LIN {X -22.647,Y -45.817,Z -234.027,A -90.000,B 90.000,C 0.000} C_DIS
LIN {X -22.412,Y -45.824,Z -234.254,A -90.000,B 90.000,C 0.000} C_DIS
LIN {X -21.688,Y -45.853,Z -235.006,A -90.000,B 90.000,C 0.000} C_DIS
LIN {X -21.666,Y -45.854,Z -235.029,A -90.000,B 90.000,C 0.000} C_DIS
LIN {X -21.383,Y -45.849,Z -235.328,A -90.000,B 90.000,C 0.000} C_DIS
LIN {X -21.097,Y -45.839,Z -235.634,A -90.000,B 90.000,C 0.000} C_DIS
LIN {X -20.891,Y -45.833,Z -235.870,A -90.000,B 90.000,C 0.000} C_DIS
LIN {X -20.670,Y -45.827,Z -236.134,A -90.000,B 90.000,C 0.000} C_DIS
LIN {X -19.793,Y -45.811,Z -237.253,A -90.000,B 90.000,C 0.000} C_DIS
LIN {X -19.564,Y -45.803,Z -237.550,A -90.000,B 90.000,C 0.000} C_DIS
LIN {X -19.412,Y -45.797,Z -237.759,A -90.000,B 90.000,C 0.000} C_DIS
LIN {X -19.249,Y -45.792,Z -237.998,A -90.000,B 90.000,C 0.000} C_DIS
LIN {X -19.122,Y -45.789,Z -238.198,A -90.000,B 90.000,C 0.000} C_DIS
LIN {X -19.022,Y -45.787,Z -238.366,A -90.000,B 90.000,C 0.000} C_DIS
LIN {X -18.604,Y -45.783,Z -239.120,A -90.000,B 90.000,C 0.000} C_DIS
LIN {X -18.544,Y -45.783,Z -239.238,A -90.000,B 90.000,C 0.000} C_DIS
LIN {X -18.361,Y -45.785,Z -239.635,A -90.000,B 90.000,C 0.000} C_DIS
LIN {X -18.257,Y -45.789,Z -239.886,A -90.000,B 90.000,C 0.000} C_DIS
LIN {X -18.034,Y -45.806,Z -240.496,A -90.000,B 90.000,C 0.000} C_DIS
LIN {X -17.944,Y -45.815,Z -240.763,A -90.000,B 90.000,C 0.000} C_DIS
LIN {X -17.916,Y -45.818,Z -240.851,A -90.000,B 90.000,C 0.000} C_DIS
LIN {X -17.863,Y -45.826,Z -241.042,A -90.000,B 90.000,C 0.000} C_DIS
LIN {X -17.792,Y -45.839,Z -241.338,A -90.000,B 90.000,C 0.000} C_DIS
LIN {X -17.768,Y -45.845,Z -241.457,A -90.000,B 90.000,C 0.000} C_DIS
LIN {X -17.629,Y -45.884,Z -242.163,A -90.000,B 90.000,C 0.000} C_DIS
LIN {X -17.582,Y -45.904,Z -242.488,A -90.000,B 90.000,C 0.000} C_DIS
LIN {X -17.534,Y -45.934,Z -242.926,A -90.000,B 90.000,C 0.000} C_DIS
LIN {X -17.511,Y -45.957,Z -243.232,A -90.000,B 90.000,C 0.000} C_DIS
LIN {X -17.499,Y -45.988,Z -243.561,A -90.000,B 90.000,C 0.000} C_DIS
LIN {X -17.499,Y -60.000,Z -243.561,A -90.000,B 90.000,C 0.000} C_DIS
LIN {X -25.308,Y -60.000,Z -229.853,A -90.000,B 90.000,C 0.000} C_DIS
LIN {X -25.308,Y -45.308,Z -229.853,A -90.000,B 90.000,C 0.000} C_DIS
LIN {X -25.272,Y -45.313,Z -229.872,A -90.000,B 90.000,C 0.000} C_DIS
LIN {X -25.025,Y -45.335,Z -230.008,A -90.000,B 90.000,C 0.000} C_DIS
LIN {X -24.905,Y -45.346,Z -230.078,A -90.000,B 90.000,C 0.000} C_DIS
LIN {X -23.343,Y -45.449,Z -231.019,A -90.000,B 90.000,C 0.000} C_DIS
LIN {X -22.863,Y -45.483,Z -231.328,A -90.000,B 90.000,C 0.000} C_DIS
LIN {X -22.629,Y -45.500,Z -231.488,A -90.000,B 90.000,C 0.000} C_DIS
LIN {X -22.520,Y -45.509,Z -231.567,A -90.000,B 90.000,C 0.000} C_DIS
LIN {X -22.280,Y -45.526,Z -231.743,A -90.000,B 90.000,C 0.000} C_DIS
LIN {X -21.917,Y -45.530,Z -232.035,A -90.000,B 90.000,C 0.000} C_DIS
LIN {X -21.614,Y -45.534,Z -232.290,A -90.000,B 90.000,C 0.000} C_DIS
LIN {X -21.315,Y -45.541,Z -232.561,A -90.000,B 90.000,C 0.000} C_DIS
LIN {X -21.031,Y -45.549,Z -232.834,A -90.000,B 90.000,C 0.000} C_DIS
LIN {X -20.941,Y -45.552,Z -232.926,A -90.000,B 90.000,C 0.000} C_DIS
LIN {X -20.117,Y -45.581,Z -233.783,A -90.000,B 90.000,C 0.000} C_DIS
LIN {X -20.016,Y -45.579,Z -233.890,A -90.000,B 90.000,C 0.000} C_DIS
LIN {X -19.653,Y -45.565,Z -234.278,A -90.000,B 90.000,C 0.000} C_DIS
LIN {X -19.404,Y -45.557,Z -234.562,A -90.000,B 90.000,C 0.000} C_DIS
LIN {X -19.155,Y -45.549,Z -234.858,A -90.000,B 90.000,C 0.000} C_DIS
LIN {X -18.235,Y -45.525,Z -236.032,A -90.000,B 90.000,C 0.000} C_DIS
LIN {X -18.007,Y -45.513,Z -236.330,A -90.000,B 90.000,C 0.000} C_DIS
LIN {X -17.818,Y -45.504,Z -236.588,A -90.000,B 90.000,C 0.000} C_DIS
LIN {X -17.619,Y -45.495,Z -236.878,A -90.000,B 90.000,C 0.000} C_DIS
LIN {X -17.455,Y -45.489,Z -237.133,A -90.000,B 90.000,C 0.000} C_DIS
LIN {X -17.326,Y -45.485,Z -237.350,A -90.000,B 90.000,C 0.000} C_DIS
LIN {X -16.875,Y -45.480,Z -238.161,A -90.000,B 90.000,C 0.000} C_DIS
LIN {X -16.778,Y -45.480,Z -238.349,A -90.000,B 90.000,C 0.000} C_DIS
LIN {X -16.681,Y -45.481,Z -238.557,A -90.000,B 90.000,C 0.000} C_DIS
LIN {X -16.533,Y -45.487,Z -238.879,A -90.000,B 90.000,C 0.000} C_DIS
LIN {X -16.428,Y -45.494,Z -239.131,A -90.000,B 90.000,C 0.000} C_DIS
LIN {X -16.395,Y -45.497,Z -239.215,A -90.000,B 90.000,C 0.000} C_DIS
LIN {X -16.172,Y -45.519,Z -239.825,A -90.000,B 90.000,C 0.000} C_DIS
LIN {X -16.066,Y -45.531,Z -240.136,A -90.000,B 90.000,C 0.000} C_DIS
LIN {X -16.020,Y -45.538,Z -240.280,A -90.000,B 90.000,C 0.000} C_DIS
LIN {X -15.949,Y -45.549,Z -240.529,A -90.000,B 90.000,C 0.000} C_DIS
LIN {X -15.847,Y -45.571,Z -240.957,A -90.000,B 90.000,C 0.000} C_DIS
LIN {X -15.723,Y -45.607,Z -241.586,A -90.000,B 90.000,C 0.000} C_DIS
LIN {X -15.681,Y -45.623,Z -241.796,A -90.000,B 90.000,C 0.000} C_DIS
LIN {X -15.664,Y -45.631,Z -241.894,A -90.000,B 90.000,C 0.000} C_DIS
LIN {X -15.616,Y -45.658,Z -242.218,A -90.000,B 90.000,C 0.000} C_DIS
LIN {X -15.558,Y -45.701,Z -242.722,A -90.000,B 90.000,C 0.000} C_DIS
LIN {X -15.527,Y -45.736,Z -243.100,A -90.000,B 90.000,C 0.000} C_DIS
LIN {X -15.523,Y -45.743,Z -243.182,A -90.000,B 90.000,C 0.000} C_DIS
LIN {X -15.510,Y -45.779,Z -243.561,A -90.000,B 90.000,C 0.000} C_DIS
LIN {X -15.498,Y -45.807,Z -243.852,A -90.000,B 90.000,C 0.000} C_DIS
LIN {X -15.490,Y -45.818,Z -243.968,A -90.000,B 90.000,C 0.000} C_DIS
LIN {X -15.473,Y -45.834,Z -244.149,A -90.000,B 90.000,C 0.000} C_DIS
LIN {X -15.463,Y -45.839,Z -244.213,A -90.000,B 90.000,C 0.000} C_DIS
LIN {X -15.448,Y -45.845,Z -244.280,A -90.000,B 90.000,C 0.000} C_DIS
LIN {X -15.436,Y -45.846,Z -244.306,A -90.000,B 90.000,C 0.000} C_DIS
LIN {X -15.430,Y -45.847,Z -244.313,A -90.000,B 90.000,C 0.000} C_DIS
LIN {X -15.417,Y -45.846,Z -244.317,A -90.000,B 90.000,C 0.000} C_DIS
LIN {X -15.404,Y -45.844,Z -244.307,A -90.000,B 90.000,C 0.000} C_DIS
LIN {X -15.390,Y -45.840,Z -244.284,A -90.000,B 90.000,C 0.000} C_DIS
LIN {X -15.360,Y -45.829,Z -244.201,A -90.000,B 90.000,C 0.000} C_DIS
LIN {X -15.328,Y -45.813,Z -244.074,A -90.000,B 90.000,C 0.000} C_DIS
LIN {X -15.293,Y -45.792,Z -243.906,A -90.000,B 90.000,C 0.000} C_DIS
LIN {X -15.215,Y -45.740,Z -243.472,A -90.000,B 90.000,C 0.000} C_DIS
LIN {X -14.980,Y -45.573,Z -242.035,A -90.000,B 90.000,C 0.000} C_DIS
LIN {X -14.871,Y -45.501,Z -241.424,A -90.000,B 90.000,C 0.000} C_DIS
LIN {X -14.814,Y -45.466,Z -241.130,A -90.000,B 90.000,C 0.000} C_DIS
LIN {X -14.755,Y -45.433,Z -240.851,A -90.000,B 90.000,C 0.000} C_DIS
LIN {X -14.694,Y -45.402,Z -240.592,A -90.000,B 90.000,C 0.000} C_DIS
LIN {X -14.632,Y -45.376,Z -240.356,A -90.000,B 90.000,C 0.000} C_DIS
LIN {X -14.568,Y -45.352,Z -240.151,A -90.000,B 90.000,C 0.000} C_DIS
LIN {X -14.502,Y -45.330,Z -239.980,A -90.000,B 90.000,C 0.000} C_DIS
LIN {X -14.469,Y -45.320,Z -239.908,A -90.000,B 90.000,C 0.000} C_DIS
LIN {X -14.435,Y -45.311,Z -239.848,A -90.000,B 90.000,C 0.000} C_DIS
LIN {X -14.401,Y -45.303,Z -239.798,A -90.000,B 90.000,C 0.000} C_DIS
LIN {X -14.367,Y -45.296,Z -239.760,A -90.000,B 90.000,C 0.000} C_DIS
LIN {X -14.332,Y -45.290,Z -239.734,A -90.000,B 90.000,C 0.000} C_DIS
LIN {X -14.297,Y -45.284,Z -239.722,A -90.000,B 90.000,C 0.000} C_DIS
LIN {X -14.262,Y -45.280,Z -239.723,A -90.000,B 90.000,C 0.000} C_DIS
LIN {X -14.244,Y -45.278,Z -239.728,A -90.000,B 90.000,C 0.000} C_DIS
LIN {X -14.208,Y -45.276,Z -239.751,A -90.000,B 90.000,C 0.000} C_DIS
LIN {X -14.172,Y -45.275,Z -239.788,A -90.000,B 90.000,C 0.000} C_DIS
LIN {X -14.136,Y -45.274,Z -239.841,A -90.000,B 90.000,C 0.000} C_DIS
LIN {X -14.118,Y -45.275,Z -239.874,A -90.000,B 90.000,C 0.000} C_DIS
LIN {X -14.062,Y -45.278,Z -239.997,A -90.000,B 90.000,C 0.000} C_DIS
LIN {X -14.025,Y -45.282,Z -240.101,A -90.000,B 90.000,C 0.000} C_DIS
LIN {X -13.988,Y -45.290,Z -240.223,A -90.000,B 90.000,C 0.000} C_DIS
LIN {X -13.931,Y -45.308,Z -240.442,A -90.000,B 90.000,C 0.000} C_DIS
LIN {X -13.901,Y -45.320,Z -240.569,A -90.000,B 90.000,C 0.000} C_DIS
LIN {X -13.728,Y -45.398,Z -241.425,A -90.000,B 90.000,C 0.000} C_DIS
LIN {X -13.702,Y -45.412,Z -241.572,A -90.000,B 90.000,C 0.000} C_DIS
LIN {X -13.646,Y -45.448,Z -241.945,A -90.000,B 90.000,C 0.000} C_DIS
LIN {X -13.580,Y -45.502,Z -242.498,A -90.000,B 90.000,C 0.000} C_DIS
LIN {X -13.541,Y -45.549,Z -242.959,A -90.000,B 90.000,C 0.000} C_DIS
LIN {X -13.533,Y -45.562,Z -243.089,A -90.000,B 90.000,C 0.000} C_DIS
LIN {X -13.522,Y -45.596,Z -243.405,A -90.000,B 90.000,C 0.000} C_DIS
LIN {X -13.516,Y -45.621,Z -243.561,A -90.000,B 90.000,C 0.000} C_DIS
LIN {X -13.504,Y -45.657,Z -243.764,A -90.000,B 90.000,C 0.000} C_DIS
LIN {X -13.495,Y -45.671,Z -243.847,A -90.000,B 90.000,C 0.000} C_DIS
LIN {X -13.472,Y -45.692,Z -243.979,A -90.000,B 90.000,C 0.000} C_DIS
LIN {X -13.457,Y -45.699,Z -244.028,A -90.000,B 90.000,C 0.000} C_DIS
LIN {X -13.432,Y -45.708,Z -244.081,A -90.000,B 90.000,C 0.000} C_DIS
LIN {X -13.404,Y -45.712,Z -244.113,A -90.000,B 90.000,C 0.000} C_DIS
LIN {X -13.394,Y -45.713,Z -244.119,A -90.000,B 90.000,C 0.000} C_DIS
LIN {X -13.372,Y -45.713,Z -244.123,A -90.000,B 90.000,C 0.000} C_DIS
LIN {X -13.349,Y -45.711,Z -244.119,A -90.000,B 90.000,C 0.000} C_DIS
LIN {X -13.324,Y -45.709,Z -244.107,A -90.000,B 90.000,C 0.000} C_DIS
LIN {X -13.298,Y -45.705,Z -244.086,A -90.000,B 90.000,C 0.000} C_DIS
LIN {X -13.257,Y -45.696,Z -244.042,A -90.000,B 90.000,C 0.000} C_DIS
LIN {X -13.198,Y -45.681,Z -243.959,A -90.000,B 90.000,C 0.000} C_DIS
LIN {X -13.135,Y -45.661,Z -243.851,A -90.000,B 90.000,C 0.000} C_DIS
LIN {X -13.068,Y -45.638,Z -243.723,A -90.000,B 90.000,C 0.000} C_DIS
LIN {X -12.962,Y -45.597,Z -243.497,A -90.000,B 90.000,C 0.000} C_DIS
LIN {X -12.812,Y -45.536,Z -243.153,A -90.000,B 90.000,C 0.000} C_DIS
LIN {X -12.576,Y -45.437,Z -242.596,A -90.000,B 90.000,C 0.000} C_DIS
LIN {X -12.496,Y -45.407,Z -242.412,A -90.000,B 90.000,C 0.000} C_DIS
LIN {X -12.417,Y -45.381,Z -242.235,A -90.000,B 90.000,C 0.000} C_DIS
LIN {X -12.300,Y -45.345,Z -241.988,A -90.000,B 90.000,C 0.000} C_DIS
LIN {X -12.186,Y -45.313,Z -241.774,A -90.000,B 90.000,C 0.000} C_DIS
LIN {X -12.113,Y -45.294,Z -241.655,A -90.000,B 90.000,C 0.000} C_DIS
LIN {X -12.077,Y -45.286,Z -241.604,A -90.000,B 90.000,C 0.000} C_DIS
LIN {X -12.042,Y -45.278,Z -241.558,A -90.000,B 90.000,C 0.000} C_DIS
LIN {X -11.991,Y -45.268,Z -241.503,A -90.000,B 90.000,C 0.000} C_DIS
LIN {X -11.959,Y -45.263,Z -241.475,A -90.000,B 90.000,C 0.000} C_DIS
LIN {X -11.927,Y -45.258,Z -241.454,A -90.000,B 90.000,C 0.000} C_DIS
LIN {X -11.896,Y -45.254,Z -241.441,A -90.000,B 90.000,C 0.000} C_DIS
LIN {X -11.866,Y -45.251,Z -241.437,A -90.000,B 90.000,C 0.000} C_DIS
LIN {X -11.838,Y -45.249,Z -241.441,A -90.000,B 90.000,C 0.000} C_DIS
LIN {X -11.824,Y -45.249,Z -241.446,A -90.000,B 90.000,C 0.000} C_DIS
LIN {X -11.797,Y -45.249,Z -241.464,A -90.000,B 90.000,C 0.000} C_DIS
LIN {X -11.784,Y -45.249,Z -241.477,A -90.000,B 90.000,C 0.000} C_DIS
LIN {X -11.747,Y -45.252,Z -241.530,A -90.000,B 90.000,C 0.000} C_DIS
LIN {X -11.713,Y -45.257,Z -241.606,A -90.000,B 90.000,C 0.000} C_DIS
LIN {X -11.683,Y -45.266,Z -241.708,A -90.000,B 90.000,C 0.000} C_DIS
LIN {X -11.665,Y -45.278,Z -241.790,A -90.000,B 90.000,C 0.000} C_DIS
LIN {X -11.648,Y -45.293,Z -241.885,A -90.000,B 90.000,C 0.000} C_DIS
LIN {X -11.633,Y -45.308,Z -241.992,A -90.000,B 90.000,C 0.000} C_DIS
LIN {X -11.598,Y -45.355,Z -242.277,A -90.000,B 90.000,C 0.000} C_DIS
LIN {X -11.550,Y -45.440,Z -242.801,A -90.000,B 90.000,C 0.000} C_DIS
LIN {X -11.539,Y -45.469,Z -242.976,A -90.000,B 90.000,C 0.000} C_DIS
LIN {X -11.517,Y -45.565,Z -243.561,A -90.000,B 90.000,C 0.000} C_DIS
LIN {X -11.503,Y -45.599,Z -243.751,A -90.000,B 90.000,C 0.000} C_DIS
LIN {X -11.494,Y -45.611,Z -243.830,A -90.000,B 90.000,C 0.000} C_DIS
LIN {X -11.476,Y -45.627,Z -243.927,A -90.000,B 90.000,C 0.000} C_DIS
LIN {X -11.455,Y -45.639,Z -244.002,A -90.000,B 90.000,C 0.000} C_DIS
LIN {X -11.438,Y -45.646,Z -244.039,A -90.000,B 90.000,C 0.000} C_DIS
LIN {X -11.409,Y -45.653,Z -244.079,A -90.000,B 90.000,C 0.000} C_DIS
LIN {X -11.387,Y -45.656,Z -244.094,A -90.000,B 90.000,C 0.000} C_DIS
LIN {X -11.375,Y -45.657,Z -244.098,A -90.000,B 90.000,C 0.000} C_DIS
LIN {X -11.351,Y -45.658,Z -244.101,A -90.000,B 90.000,C 0.000} C_DIS
LIN {X -11.326,Y -45.658,Z -244.096,A -90.000,B 90.000,C 0.000} C_DIS
LIN {X -11.284,Y -45.655,Z -244.075,A -90.000,B 90.000,C 0.000} C_DIS
LIN {X -11.255,Y -45.652,Z -244.053,A -90.000,B 90.000,C 0.000} C_DIS
LIN {X -11.209,Y -45.646,Z -244.007,A -90.000,B 90.000,C 0.000} C_DIS
LIN {X -11.143,Y -45.634,Z -243.925,A -90.000,B 90.000,C 0.000} C_DIS
LIN {X -11.037,Y -45.609,Z -243.765,A -90.000,B 90.000,C 0.000} C_DIS
LIN {X -10.962,Y -45.590,Z -243.637,A -90.000,B 90.000,C 0.000} C_DIS
LIN {X -10.844,Y -45.556,Z -243.421,A -90.000,B 90.000,C 0.000} C_DIS
LIN {X -10.430,Y -45.424,Z -242.614,A -90.000,B 90.000,C 0.000} C_DIS
LIN {X -10.265,Y -45.372,Z -242.312,A -90.000,B 90.000,C 0.000} C_DIS
LIN {X -10.185,Y -45.348,Z -242.177,A -90.000,B 90.000,C 0.000} C_DIS
LIN {X -10.108,Y -45.326,Z -242.058,A -90.000,B 90.000,C 0.000} C_DIS
LIN {X -10.033,Y -45.306,Z -241.955,A -90.000,B 90.000,C 0.000} C_DIS
LIN {X -9.963,Y -45.289,Z -241.874,A -90.000,B 90.000,C 0.000} C_DIS
LIN {X -9.929,Y -45.282,Z -241.842,A -90.000,B 90.000,C 0.000} C_DIS
LIN {X -9.896,Y -45.276,Z -241.816,A -90.000,B 90.000,C 0.000} C_DIS
LIN {X -9.864,Y -45.270,Z -241.797,A -90.000,B 90.000,C 0.000} C_DIS
LIN {X -9.833,Y -45.266,Z -241.785,A -90.000,B 90.000,C 0.000} C_DIS
LIN {X -9.804,Y -45.262,Z -241.781,A -90.000,B 90.000,C 0.000} C_DIS
LIN {X -9.776,Y -45.260,Z -241.784,A -90.000,B 90.000,C 0.000} C_DIS
LIN {X -9.750,Y -45.259,Z -241.795,A -90.000,B 90.000,C 0.000} C_DIS
LIN {X -9.725,Y -45.259,Z -241.815,A -90.000,B 90.000,C 0.000} C_DIS
LIN {X -9.701,Y -45.260,Z -241.844,A -90.000,B 90.000,C 0.000} C_DIS
LIN {X -9.680,Y -45.262,Z -241.882,A -90.000,B 90.000,C 0.000} C_DIS
LIN {X -9.650,Y -45.269,Z -241.957,A -90.000,B 90.000,C 0.000} C_DIS
LIN {X -9.623,Y -45.278,Z -242.054,A -90.000,B 90.000,C 0.000} C_DIS
LIN {X -9.596,Y -45.298,Z -242.223,A -90.000,B 90.000,C 0.000} C_DIS
LIN {X -9.587,Y -45.308,Z -242.324,A -90.000,B 90.000,C 0.000} C_DIS
LIN {X -9.584,Y -45.312,Z -242.357,A -90.000,B 90.000,C 0.000} C_DIS
LIN {X -9.559,Y -45.357,Z -242.634,A -90.000,B 90.000,C 0.000} C_DIS
LIN {X -9.544,Y -45.393,Z -242.855,A -90.000,B 90.000,C 0.000} C_DIS
LIN {X -9.521,Y -45.489,Z -243.439,A -90.000,B 90.000,C 0.000} C_DIS
LIN {X -9.518,Y -45.504,Z -243.561,A -90.000,B 90.000,C 0.000} C_DIS
LIN {X -9.514,Y -45.515,Z -243.653,A -90.000,B 90.000,C 0.000} C_DIS
LIN {X -9.498,Y -45.537,Z -243.827,A -90.000,B 90.000,C 0.000} C_DIS
LIN {X -9.472,Y -45.557,Z -243.990,A -90.000,B 90.000,C 0.000} C_DIS
LIN {X -9.436,Y -45.575,Z -244.141,A -90.000,B 90.000,C 0.000} C_DIS
LIN {X -9.390,Y -45.599,Z -244.280,A -90.000,B 90.000,C 0.000} C_DIS
LIN {X -9.337,Y -45.621,Z -244.408,A -90.000,B 90.000,C 0.000} C_DIS
LIN {X -9.308,Y -45.632,Z -244.467,A -90.000,B 90.000,C 0.000} C_DIS
LIN {X -9.276,Y -45.642,Z -244.523,A -90.000,B 90.000,C 0.000} C_DIS
LIN {X -9.209,Y -45.661,Z -244.628,A -90.000,B 90.000,C 0.000} C_DIS
LIN {X -9.173,Y -45.669,Z -244.676,A -90.000,B 90.000,C 0.000} C_DIS
LIN {X -9.098,Y -45.685,Z -244.761,A -90.000,B 90.000,C 0.000} C_DIS
LIN {X -9.018,Y -45.698,Z -244.834,A -90.000,B 90.000,C 0.000} C_DIS
LIN {X -8.934,Y -45.710,Z -244.896,A -90.000,B 90.000,C 0.000} C_DIS
LIN {X -8.847,Y -45.720,Z -244.949,A -90.000,B 90.000,C 0.000} C_DIS
LIN {X -8.757,Y -45.727,Z -244.988,A -90.000,B 90.000,C 0.000} C_DIS
LIN {X -8.712,Y -45.730,Z -245.004,A -90.000,B 90.000,C 0.000} C_DIS
LIN {X -8.620,Y -45.735,Z -245.027,A -90.000,B 90.000,C 0.000} C_DIS
LIN {X -8.527,Y -45.738,Z -245.037,A -90.000,B 90.000,C 0.000} C_DIS
LIN {X -8.434,Y -45.739,Z -245.037,A -90.000,B 90.000,C 0.000} C_DIS
LIN {X -8.342,Y -45.738,Z -245.025,A -90.000,B 90.000,C 0.000} C_DIS
LIN {X -8.251,Y -45.735,Z -245.002,A -90.000,B 90.000,C 0.000} C_DIS
LIN {X -8.163,Y -45.730,Z -244.968,A -90.000,B 90.000,C 0.000} C_DIS
LIN {X -8.077,Y -45.723,Z -244.922,A -90.000,B 90.000,C 0.000} C_DIS
LIN {X -7.995,Y -45.714,Z -244.866,A -90.000,B 90.000,C 0.000} C_DIS
LIN {X -7.917,Y -45.703,Z -244.797,A -90.000,B 90.000,C 0.000} C_DIS
LIN {X -7.879,Y -45.697,Z -244.759,A -90.000,B 90.000,C 0.000} C_DIS
LIN {X -7.844,Y -45.690,Z -244.718,A -90.000,B 90.000,C 0.000} C_DIS
LIN {X -7.808,Y -45.683,Z -244.674,A -90.000,B 90.000,C 0.000} C_DIS
LIN {X -7.775,Y -45.676,Z -244.627,A -90.000,B 90.000,C 0.000} C_DIS
LIN {X -7.713,Y -45.658,Z -244.523,A -90.000,B 90.000,C 0.000} C_DIS
LIN {X -7.685,Y -45.649,Z -244.467,A -90.000,B 90.000,C 0.000} C_DIS
LIN {X -7.633,Y -45.629,Z -244.346,A -90.000,B 90.000,C 0.000} C_DIS
LIN {X -7.591,Y -45.606,Z -244.212,A -90.000,B 90.000,C 0.000} C_DIS
LIN {X -7.574,Y -45.594,Z -244.141,A -90.000,B 90.000,C 0.000} C_DIS
LIN {X -7.557,Y -45.582,Z -244.067,A -90.000,B 90.000,C 0.000} C_DIS
LIN {X -7.534,Y -45.555,Z -243.910,A -90.000,B 90.000,C 0.000} C_DIS
LIN {X -7.521,Y -45.526,Z -243.742,A -90.000,B 90.000,C 0.000} C_DIS
LIN {X -7.518,Y -45.494,Z -243.561,A -90.000,B 90.000,C 0.000} C_DIS
LIN {X -7.523,Y -45.471,Z -243.366,A -90.000,B 90.000,C 0.000} C_DIS
LIN {X -7.548,Y -45.398,Z -242.727,A -90.000,B 90.000,C 0.000} C_DIS
LIN {X -7.554,Y -45.387,Z -242.637,A -90.000,B 90.000,C 0.000} C_DIS
LIN {X -7.567,Y -45.354,Z -242.454,A -90.000,B 90.000,C 0.000} C_DIS
LIN {X -7.589,Y -45.308,Z -242.209,A -90.000,B 90.000,C 0.000} C_DIS
LIN {X -7.598,Y -45.293,Z -242.101,A -90.000,B 90.000,C 0.000} C_DIS
LIN {X -7.604,Y -45.262,Z -241.922,A -90.000,B 90.000,C 0.000} C_DIS
LIN {X -7.597,Y -45.247,Z -241.789,A -90.000,B 90.000,C 0.000} C_DIS
LIN {X -7.588,Y -45.241,Z -241.739,A -90.000,B 90.000,C 0.000} C_DIS
LIN {X -7.569,Y -45.234,Z -241.683,A -90.000,B 90.000,C 0.000} C_DIS
LIN {X -7.544,Y -45.230,Z -241.649,A -90.000,B 90.000,C 0.000} C_DIS
LIN {X -7.534,Y -45.229,Z -241.642,A -90.000,B 90.000,C 0.000} C_DIS
LIN {X -7.513,Y -45.229,Z -241.635,A -90.000,B 90.000,C 0.000} C_DIS
LIN {X -7.489,Y -45.229,Z -241.637,A -90.000,B 90.000,C 0.000} C_DIS
LIN {X -7.448,Y -45.231,Z -241.655,A -90.000,B 90.000,C 0.000} C_DIS
LIN {X -7.418,Y -45.233,Z -241.676,A -90.000,B 90.000,C 0.000} C_DIS
LIN {X -7.386,Y -45.237,Z -241.705,A -90.000,B 90.000,C 0.000} C_DIS
LIN {X -7.351,Y -45.243,Z -241.740,A -90.000,B 90.000,C 0.000} C_DIS
LIN {X -7.277,Y -45.264,Z -241.829,A -90.000,B 90.000,C 0.000} C_DIS
LIN {X -7.153,Y -45.305,Z -242.004,A -90.000,B 90.000,C 0.000} C_DIS
LIN {X -7.017,Y -45.353,Z -242.218,A -90.000,B 90.000,C 0.000} C_DIS
LIN {X -6.921,Y -45.383,Z -242.377,A -90.000,B 90.000,C 0.000} C_DIS
LIN {X -6.410,Y -45.504,Z -243.250,A -90.000,B 90.000,C 0.000} C_DIS
LIN {X -6.209,Y -45.549,Z -243.577,A -90.000,B 90.000,C 0.000} C_DIS
LIN {X -6.065,Y -45.579,Z -243.789,A -90.000,B 90.000,C 0.000} C_DIS
LIN {X -5.975,Y -45.596,Z -243.909,A -90.000,B 90.000,C 0.000} C_DIS
LIN {X -5.932,Y -45.604,Z -243.962,A -90.000,B 90.000,C 0.000} C_DIS
LIN {X -5.851,Y -45.617,Z -244.050,A -90.000,B 90.000,C 0.000} C_DIS
LIN {X -5.813,Y -45.622,Z -244.084,A -90.000,B 90.000,C 0.000} C_DIS
LIN {X -5.776,Y -45.627,Z -244.112,A -90.000,B 90.000,C 0.000} C_DIS
LIN {X -5.742,Y -45.631,Z -244.132,A -90.000,B 90.000,C 0.000} C_DIS
LIN {X -5.709,Y -45.633,Z -244.145,A -90.000,B 90.000,C 0.000} C_DIS
LIN {X -5.679,Y -45.635,Z -244.150,A -90.000,B 90.000,C 0.000} C_DIS
LIN {X -5.665,Y -45.636,Z -244.149,A -90.000,B 90.000,C 0.000} C_DIS
LIN {X -5.638,Y -45.636,Z -244.141,A -90.000,B 90.000,C 0.000} C_DIS
LIN {X -5.625,Y -45.635,Z -244.134,A -90.000,B 90.000,C 0.000} C_DIS
LIN {X -5.602,Y -45.634,Z -244.113,A -90.000,B 90.000,C 0.000} C_DIS
LIN {X -5.591,Y -45.633,Z -244.098,A -90.000,B 90.000,C 0.000} C_DIS
LIN {X -5.563,Y -45.627,Z -244.040,A -90.000,B 90.000,C 0.000} C_DIS
LIN {X -5.542,Y -45.619,Z -243.959,A -90.000,B 90.000,C 0.000} C_DIS
LIN {X -5.527,Y -45.608,Z -243.853,A -90.000,B 90.000,C 0.000} C_DIS
LIN {X -5.519,Y -45.587,Z -243.671,A -90.000,B 90.000,C 0.000} C_DIS
LIN {X -5.520,Y -45.574,Z -243.561,A -90.000,B 90.000,C 0.000} C_DIS
LIN {X -5.526,Y -45.542,Z -243.274,A -90.000,B 90.000,C 0.000} C_DIS
LIN {X -5.554,Y -45.462,Z -242.581,A -90.000,B 90.000,C 0.000} C_DIS
LIN {X -5.580,Y -45.422,Z -242.237,A -90.000,B 90.000,C 0.000} C_DIS
LIN {X -5.609,Y -45.387,Z -241.939,A -90.000,B 90.000,C 0.000} C_DIS
LIN {X -5.642,Y -45.352,Z -241.754,A -90.000,B 90.000,C 0.000} C_DIS
LIN {X -5.662,Y -45.337,Z -241.677,A -90.000,B 90.000,C 0.000} C_DIS
LIN {X -5.686,Y -45.321,Z -241.596,A -90.000,B 90.000,C 0.000} C_DIS
LIN {X -5.707,Y -45.308,Z -241.534,A -90.000,B 90.000,C 0.000} C_DIS
LIN {X -5.707,Y -60.000,Z -241.534,A -90.000,B 90.000,C 0.000} C_DIS
LIN {X -18.858,Y -60.000,Z -232.233,A -90.000,B 90.000,C 0.000} C_DIS
LIN {X -18.858,Y -45.308,Z -232.233,A -90.000,B 90.000,C 0.000} C_DIS
LIN {X -18.568,Y -45.317,Z -232.535,A -90.000,B 90.000,C 0.000} C_DIS
LIN {X -18.401,Y -45.314,Z -232.714,A -90.000,B 90.000,C 0.000} C_DIS
LIN {X -18.264,Y -45.308,Z -232.861,A -90.000,B 90.000,C 0.000} C_DIS
LIN {X -18.264,Y -60.000,Z -232.861,A -90.000,B 90.000,C 0.000} C_DIS
LIN {X -62.179,Y -60.000,Z -243.561,A -90.000,B 90.000,C 0.000} C_DIS
LIN {X -62.179,Y -46.130,Z -243.561,A -90.000,B 90.000,C 0.000} C_DIS
LIN {X -62.165,Y -46.075,Z -243.443,A -90.000,B 90.000,C 0.000} C_DIS
LIN {X -62.138,Y -45.979,Z -243.241,A -90.000,B 90.000,C 0.000} C_DIS
LIN {X -62.094,Y -45.870,Z -243.007,A -90.000,B 90.000,C 0.000} C_DIS
LIN {X -62.018,Y -45.731,Z -242.700,A -90.000,B 90.000,C 0.000} C_DIS
LIN {X -61.986,Y -45.680,Z -242.586,A -90.000,B 90.000,C 0.000} C_DIS
LIN {X -61.922,Y -45.595,Z -242.389,A -90.000,B 90.000,C 0.000} C_DIS
LIN {X -61.847,Y -45.507,Z -242.181,A -90.000,B 90.000,C 0.000} C_DIS
LIN {X -61.779,Y -45.437,Z -242.012,A -90.000,B 90.000,C 0.000} C_DIS
LIN {X -61.681,Y -45.348,Z -241.792,A -90.000,B 90.000,C 0.000} C_DIS
LIN {X -61.629,Y -45.308,Z -241.691,A -90.000,B 90.000,C 0.000} C_DIS
LIN {X -61.522,Y -45.225,Z -241.471,A -90.000,B 90.000,C 0.000} C_DIS
LIN {X -61.414,Y -45.135,Z -241.245,A -90.000,B 90.000,C 0.000} C_DIS
LIN {X -61.378,Y -45.099,Z -241.156,A -90.000,B 90.000,C 0.000} C_DIS
LIN {X -61.369,Y -45.082,Z -241.119,A -90.000,B 90.000,C 0.000} C_DIS
LIN {X -61.369,Y -45.078,Z -241.112,A -90.000,B 90.000,C 0.000} C_DIS
LIN {X -61.373,Y -45.074,Z -241.106,A -90.000,B 90.000,C 0.000} C_DIS
LIN {X -61.382,Y -45.074,Z -241.110,A -90.000,B 90.000,C 0.000} C_DIS
LIN {X -61.399,Y -45.076,Z -241.123,A -90.000,B 90.000,C 0.000} C_DIS
LIN {X -61.419,Y -45.083,Z -241.146,A -90.000,B 90.000,C 0.000} C_DIS
LIN {X -61.511,Y -45.120,Z -241.263,A -90.000,B 90.000,C 0.000} C_DIS
LIN {X -61.695,Y -45.206,Z -241.519,A -90.000,B 90.000,C 0.000} C_DIS
LIN {X -62.213,Y -45.459,Z -242.260,A -90.000,B 90.000,C 0.000} C_DIS
LIN {X -62.519,Y -45.602,Z -242.686,A -90.000,B 90.000,C 0.000} C_DIS
LIN {X -62.835,Y -45.742,Z -243.111,A -90.000,B 90.000,C 0.000} C_DIS
LIN {X -62.992,Y -45.804,Z -243.313,A -90.000,B 90.000,C 0.000} C_DIS
LIN {X -63.147,Y -45.859,Z -243.504,A -90.000,B 90.000,C 0.000} C_DIS
LIN {X -63.368,Y -45.929,Z -243.762,A -90.000,B 90.000,C 0.000} C_DIS
LIN {X -63.439,Y -45.948,Z -243.837,A -90.000,B 90.000,C 0.000} C_DIS
LIN {X -63.574,Y -45.981,Z -243.972,A -90.000,B 90.000,C 0.000} C_DIS
LIN {X -63.698,Y -46.003,Z -244.081,A -90.000,B 90.000,C 0.000} C_DIS
LIN {X -63.727,Y -46.006,Z -244.103,A -90.000,B 90.000,C 0.000} C_DIS
LIN {X -63.784,Y -46.011,Z -244.142,A -90.000,B 90.000,C 0.000} C_DIS
LIN {X -63.861,Y -46.012,Z -244.186,A -90.000,B 90.000,C 0.000} C_DIS
LIN {X -63.909,Y -46.009,Z -244.203,A -90.000,B 90.000,C 0.000} C_DIS
LIN {X -63.931,Y -46.006,Z -244.209,A -90.000,B 90.000,C 0.000} C_DIS
LIN {X -63.952,Y -46.002,Z -244.211,A -90.000,B 90.000,C 0.000} C_DIS
LIN {X -63.991,Y -45.992,Z -244.212,A -90.000,B 90.000,C 0.000} C_DIS
LIN {X -64.009,Y -45.985,Z -244.207,A -90.000,B 90.000,C 0.000} C_DIS
LIN {X -64.042,Y -45.969,Z -244.192,A -90.000,B 90.000,C 0.000} C_DIS
LIN {X -64.070,Y -45.948,Z -244.164,A -90.000,B 90.000,C 0.000} C_DIS
LIN {X -64.095,Y -45.922,Z -244.125,A -90.000,B 90.000,C 0.000} C_DIS
LIN {X -64.115,Y -45.891,Z -244.073,A -90.000,B 90.000,C 0.000} C_DIS
LIN {X -64.131,Y -45.856,Z -244.010,A -90.000,B 90.000,C 0.000} C_DIS
LIN {X -64.135,Y -45.838,Z -243.976,A -90.000,B 90.000,C 0.000} C_DIS
LIN {X -64.140,Y -45.795,Z -243.893,A -90.000,B 90.000,C 0.000} C_DIS
LIN {X -64.139,Y -45.748,Z -243.797,A -90.000,B 90.000,C 0.000} C_DIS
LIN {X -64.127,Y -45.666,Z -243.625,A -90.000,B 90.000,C 0.000} C_DIS
LIN {X -64.116,Y -45.631,Z -243.561,A -90.000,B 90.000,C 0.000} C_DIS
LIN {X -64.067,Y -45.456,Z -243.183,A -90.000,B 90.000,C 0.000} C_DIS
LIN {X -64.007,Y -45.308,Z -242.854,A -90.000,B 90.000,C 0.000} C_DIS
LIN {X -63.998,Y -45.286,Z -242.792,A -90.000,B 90.000,C 0.000} C_DIS
LIN {X -63.993,Y -45.260,Z -242.737,A -90.000,B 90.000,C 0.000} C_DIS
LIN {X -63.992,Y -45.235,Z -242.687,A -90.000,B 90.000,C 0.000} C_DIS
LIN {X -63.999,Y -45.201,Z -242.622,A -90.000,B 90.000,C 0.000} C_DIS
LIN {X -64.015,Y -45.170,Z -242.570,A -90.000,B 90.000,C 0.000} C_DIS
LIN {X -64.039,Y -45.142,Z -242.529,A -90.000,B 90.000,C 0.000} C_DIS
LIN {X -64.071,Y -45.119,Z -242.498,A -90.000,B 90.000,C 0.000} C_DIS
LIN {X -64.110,Y -45.099,Z -242.478,A -90.000,B 90.000,C 0.000} C_DIS
LIN {X -64.140,Y -45.087,Z -242.470,A -90.000,B 90.000,C 0.000} C_DIS
LIN {X -64.172,Y -45.077,Z -242.466,A -90.000,B 90.000,C 0.000} C_DIS
LIN {X -64.226,Y -45.065,Z -242.467,A -90.000,B 90.000,C 0.000} C_DIS
LIN {X -64.264,Y -45.058,Z -242.473,A -90.000,B 90.000,C 0.000} C_DIS
LIN {X -64.347,Y -45.048,Z -242.494,A -90.000,B 90.000,C 0.000} C_DIS
LIN {X -64.438,Y -45.042,Z -242.528,A -90.000,B 90.000,C 0.000} C_DIS
LIN {X -64.534,Y -45.039,Z -242.573,A -90.000,B 90.000,C 0.000} C_DIS
LIN {X -64.634,Y -45.041,Z -242.628,A -90.000,B 90.000,C 0.000} C_DIS
LIN {X -64.738,Y -45.045,Z -242.690,A -90.000,B 90.000,C 0.000} C_DIS
LIN {X -64.843,Y -45.053,Z -242.760,A -90.000,B 90.000,C 0.000} C_DIS
LIN {X -65.000,Y -45.069,Z -242.875,A -90.000,B 90.000,C 0.000} C_DIS
LIN {X -65.103,Y -45.082,Z -242.955,A -90.000,B 90.000,C 0.000} C_DIS
LIN {X -65.203,Y -45.098,Z -243.038,A -90.000,B 90.000,C 0.000} C_DIS
LIN {X -65.298,Y -45.114,Z -243.122,A -90.000,B 90.000,C 0.000} C_DIS
LIN {X -65.468,Y -45.151,Z -243.284,A -90.000,B 90.000,C 0.000} C_DIS
LIN {X -65.574,Y -45.180,Z -243.398,A -90.000,B 90.000,C 0.000} C_DIS
LIN {X -65.655,Y -45.209,Z -243.498,A -90.000,B 90.000,C 0.000} C_DIS
LIN {X -65.707,Y -45.236,Z -243.580,A -90.000,B 90.000,C 0.000} C_DIS
LIN {X -65.723,Y -45.253,Z -243.623,A -90.000,B 90.000,C 0.000} C_DIS
LIN {X -65.725,Y -45.265,Z -243.648,A -90.000,B 90.000,C 0.000} C_DIS
LIN {X -65.716,Y -45.276,Z -243.666,A -90.000,B 90.000,C 0.000} C_DIS
LIN {X -65.698,Y -45.286,Z -243.676,A -90.000,B 90.000,C 0.000} C_DIS
LIN {X -65.668,Y -45.295,Z -243.678,A -90.000,B 90.000,C 0.000} C_DIS
LIN {X -65.610,Y -45.304,Z -243.667,A -90.000,B 90.000,C 0.000} C_DIS
LIN {X -65.531,Y -45.311,Z -243.639,A -90.000,B 90.000,C 0.000} C_DIS
LIN {X -65.428,Y -45.314,Z -243.592,A -90.000,B 90.000,C 0.000} C_DIS
LIN {X -65.367,Y -45.308,Z -243.561,A -90.000,B 90.000,C 0.000} C_DIS
LIN {X -63.626,Y -45.308,Z -242.657,A -90.000,B 90.000,C 0.000} C_DIS
LIN {X -56.661,Y -45.308,Z -239.287,A -90.000,B 90.000,C 0.000} C_DIS
LIN {X -55.137,Y -45.308,Z -238.546,A -90.000,B 90.000,C 0.000} C_DIS
LIN {X -54.677,Y -45.308,Z -238.333,A -90.000,B 90.000,C 0.000} C_DIS
LIN {X -53.969,Y -45.308,Z -238.017,A -90.000,B 90.000,C 0.000} C_DIS
LIN {X -52.056,Y -45.308,Z -237.178,A -90.000,B 90.000,C 0.000} C_DIS
LIN {X -48.568,Y -45.308,Z -235.753,A -90.000,B 90.000,C 0.000} C_DIS
LIN {X -43.548,Y -45.308,Z -233.812,A -90.000,B 90.000,C 0.000} C_DIS
LIN {X -40.675,Y -45.308,Z -232.778,A -90.000,B 90.000,C 0.000} C_DIS
LIN {X -39.354,Y -45.308,Z -232.340,A -90.000,B 90.000,C 0.000} C_DIS
LIN {X -39.084,Y -45.308,Z -232.259,A -90.000,B 90.000,C 0.000} C_DIS
LIN {X -38.129,Y -45.308,Z -231.997,A -90.000,B 90.000,C 0.000} C_DIS
LIN {X -36.952,Y -45.308,Z -231.709,A -90.000,B 90.000,C 0.000} C_DIS
LIN {X -33.841,Y -45.308,Z -230.903,A -90.000,B 90.000,C 0.000} C_DIS
LIN {X -31.637,Y -45.308,Z -230.395,A -90.000,B 90.000,C 0.000} C_DIS
LIN {X -30.557,Y -45.308,Z -230.194,A -90.000,B 90.000,C 0.000} C_DIS
LIN {X -29.392,Y -45.308,Z -230.092,A -90.000,B 90.000,C 0.000} C_DIS
LIN {X -26.930,Y -45.308,Z -229.970,A -90.000,B 90.000,C 0.000} C_DIS
LIN {X -25.915,Y -45.308,Z -229.883,A -90.000,B 90.000,C 0.000} C_DIS
LIN {X -25.450,Y -45.308,Z -229.854,A -90.000,B 90.000,C 0.000} C_DIS
LIN {X -25.212,Y -45.308,Z -229.852,A -90.000,B 90.000,C 0.000} C_DIS
LIN {X -24.631,Y -45.308,Z -229.900,A -90.000,B 90.000,C 0.000} C_DIS
LIN {X -22.420,Y -45.308,Z -230.350,A -90.000,B 90.000,C 0.000} C_DIS
LIN {X -21.138,Y -45.308,Z -230.656,A -90.000,B 90.000,C 0.000} C_DIS
LIN {X -20.967,Y -45.308,Z -230.712,A -90.000,B 90.000,C 0.000} C_DIS
LIN {X -20.819,Y -45.308,Z -230.813,A -90.000,B 90.000,C 0.000} C_DIS
LIN {X -19.575,Y -45.308,Z -231.692,A -90.000,B 90.000,C 0.000} C_DIS
LIN {X -18.522,Y -45.308,Z -232.486,A -90.000,B 90.000,C 0.000} C_DIS
LIN {X -18.407,Y -45.308,Z -232.623,A -90.000,B 90.000,C 0.000} C_DIS
LIN {X -17.499,Y -45.308,Z -234.121,A -90.000,B 90.000,C 0.000} C_DIS
LIN {X -16.963,Y -45.308,Z -235.030,A -90.000,B 90.000,C 0.000} C_DIS
LIN {X -15.883,Y -45.308,Z -237.442,A -90.000,B 90.000,C 0.000} C_DIS
LIN {X -15.735,Y -45.308,Z -237.746,A -90.000,B 90.000,C 0.000} C_DIS
LIN {X -14.928,Y -45.308,Z -239.075,A -90.000,B 90.000,C 0.000} C_DIS
LIN {X -14.157,Y -45.308,Z -240.234,A -90.000,B 90.000,C 0.000} C_DIS
LIN {X -14.033,Y -45.308,Z -240.367,A -90.000,B 90.000,C 0.000} C_DIS
LIN {X -11.897,Y -45.308,Z -241.947,A -90.000,B 90.000,C 0.000} C_DIS
LIN {X -9.680,Y -45.308,Z -242.323,A -90.000,B 90.000,C 0.000} C_DIS
LIN {X -7.933,Y -45.308,Z -242.332,A -90.000,B 90.000,C 0.000} C_DIS
LIN {X -1.508,Y -45.308,Z -240.030,A -90.000,B 90.000,C 0.000} C_DIS
LIN {X -1.292,Y -45.308,Z -239.907,A -90.000,B 90.000,C 0.000} C_DIS
LIN {X 1.289,Y -45.308,Z -237.704,A -90.000,B 90.000,C 0.000} C_DIS
LIN {X 2.598,Y -45.308,Z -236.636,A -90.000,B 90.000,C 0.000} C_DIS
LIN {X 3.005,Y -45.308,Z -236.156,A -90.000,B 90.000,C 0.000} C_DIS
LIN {X 5.925,Y -45.308,Z -232.690,A -90.000,B 90.000,C 0.000} C_DIS
LIN {X 6.445,Y -45.308,Z -231.926,A -90.000,B 90.000,C 0.000} C_DIS
LIN {X 8.967,Y -45.308,Z -228.177,A -90.000,B 90.000,C 0.000} C_DIS
LIN {X 9.483,Y -45.308,Z -227.431,A -90.000,B 90.000,C 0.000} C_DIS
LIN {X 9.577,Y -45.308,Z -227.287,A -90.000,B 90.000,C 0.000} C_DIS
LIN {X 12.263,Y -45.308,Z -222.848,A -90.000,B 90.000,C 0.000} C_DIS
LIN {X 13.855,Y -45.308,Z -220.017,A -90.000,B 90.000,C 0.000} C_DIS
LIN {X 14.859,Y -45.308,Z -218.291,A -90.000,B 90.000,C 0.000} C_DIS
LIN {X 15.792,Y -45.308,Z -216.511,A -90.000,B 90.000,C 0.000} C_DIS
LIN {X 17.214,Y -45.308,Z -213.696,A -90.000,B 90.000,C 0.000} C_DIS
LIN {X 17.523,Y -45.308,Z -213.048,A -90.000,B 90.000,C 0.000} C_DIS
LIN {X 18.164,Y -45.308,Z -211.529,A -90.000,B 90.000,C 0.000} C_DIS
LIN {X 18.896,Y -45.308,Z -209.777,A -90.000,B 90.000,C 0.000} C_DIS
LIN {X 19.199,Y -45.308,Z -209.018,A -90.000,B 90.000,C 0.000} C_DIS
LIN {X 19.991,Y -45.308,Z -206.726,A -90.000,B 90.000,C 0.000} C_DIS
LIN {X 20.606,Y -45.308,Z -204.669,A -90.000,B 90.000,C 0.000} C_DIS
LIN {X 20.756,Y -45.308,Z -204.093,A -90.000,B 90.000,C 0.000} C_DIS
LIN {X 20.907,Y -45.308,Z -203.280,A -90.000,B 90.000,C 0.000} C_DIS
LIN {X 21.522,Y -45.308,Z -200.221,A -90.000,B 90.000,C 0.000} C_DIS
LIN {X 22.089,Y -45.308,Z -197.268,A -90.000,B 90.000,C 0.000} C_DIS
LIN {X 22.411,Y -45.308,Z -196.015,A -90.000,B 90.000,C 0.000} C_DIS
LIN {X 22.480,Y -45.308,Z -195.788,A -90.000,B 90.000,C 0.000} C_DIS
LIN {X 22.884,Y -45.308,Z -194.622,A -90.000,B 90.000,C 0.000} C_DIS
LIN {X 23.697,Y -45.308,Z -192.046,A -90.000,B 90.000,C 0.000} C_DIS
LIN {X 23.769,Y -45.308,Z -191.870,A -90.000,B 90.000,C 0.000} C_DIS
LIN {X 23.805,Y -45.308,Z -191.785,A -90.000,B 90.000,C 0.000} C_DIS
LIN {X 24.790,Y -45.308,Z -189.677,A -90.000,B 90.000,C 0.000} C_DIS
LIN {X 25.350,Y -45.308,Z -188.352,A -90.000,B 90.000,C 0.000} C_DIS
LIN {X 25.887,Y -45.308,Z -187.463,A -90.000,B 90.000,C 0.000} C_DIS
LIN {X 26.040,Y -45.308,Z -187.226,A -90.000,B 90.000,C 0.000} C_DIS
LIN {X 27.371,Y -45.308,Z -185.203,A -90.000,B 90.000,C 0.000} C_DIS
LIN {X 28.317,Y -45.308,Z -183.934,A -90.000,B 90.000,C 0.000} C_DIS
LIN {X 29.321,Y -45.308,Z -182.660,A -90.000,B 90.000,C 0.000} C_DIS
LIN {X 31.153,Y -45.308,Z -180.413,A -90.000,B 90.000,C 0.000} C_DIS
LIN {X 33.063,Y -45.308,Z -178.190,A -90.000,B 90.000,C 0.000} C_DIS
LIN {X 33.820,Y -45.308,Z -177.103,A -90.000,B 90.000,C 0.000} C_DIS
LIN {X 34.560,Y -45.308,Z -176.105,A -90.000,B 90.000,C 0.000} C_DIS
LIN {X 35.449,Y -45.308,Z -174.663,A -90.000,B 90.000,C 0.000} C_DIS
LIN {X 35.598,Y -45.308,Z -174.431,A -90.000,B 90.000,C 0.000} C_DIS
LIN {X 35.832,Y -45.308,Z -174.076,A -90.000,B 90.000,C 0.000} C_DIS
LIN {X 36.993,Y -45.308,Z -172.032,A -90.000,B 90.000,C 0.000} C_DIS
LIN {X 37.128,Y -45.308,Z -171.809,A -90.000,B 90.000,C 0.000} C_DIS
LIN {X 37.889,Y -45.308,Z -170.415,A -90.000,B 90.000,C 0.000} C_DIS
LIN {X 38.442,Y -45.308,Z -169.462,A -90.000,B 90.000,C 0.000} C_DIS
LIN {X 38.669,Y -45.308,Z -169.035,A -90.000,B 90.000,C 0.000} C_DIS
LIN {X 40.129,Y -45.308,Z -166.480,A -90.000,B 90.000,C 0.000} C_DIS
LIN {X 40.805,Y -45.308,Z -165.218,A -90.000,B 90.000,C 0.000} C_DIS
LIN {X 41.816,Y -45.308,Z -163.437,A -90.000,B 90.000,C 0.000} C_DIS
LIN {X 43.235,Y -45.308,Z -160.814,A -90.000,B 90.000,C 0.000} C_DIS
LIN {X 43.549,Y -45.308,Z -160.260,A -90.000,B 90.000,C 0.000} C_DIS
LIN {X 44.216,Y -45.308,Z -159.055,A -90.000,B 90.000,C 0.000} C_DIS
LIN {X 45.395,Y -45.308,Z -157.065,A -90.000,B 90.000,C 0.000} C_DIS
LIN {X 46.025,Y -45.308,Z -156.031,A -90.000,B 90.000,C 0.000} C_DIS
LIN {X 47.325,Y -45.308,Z -153.943,A -90.000,B 90.000,C 0.000} C_DIS
LIN {X 47.477,Y -45.308,Z -153.706,A -90.000,B 90.000,C 0.000} C_DIS
LIN {X 49.579,Y -45.308,Z -150.607,A -90.000,B 90.000,C 0.000} C_DIS
LIN {X 49.597,Y -45.308,Z -150.583,A -90.000,B 90.000,C 0.000} C_DIS
LIN {X 52.360,Y -45.308,Z -147.470,A -90.000,B 90.000,C 0.000} C_DIS
LIN {X 52.552,Y -45.308,Z -147.264,A -90.000,B 90.000,C 0.000} C_DIS
LIN {X 53.626,Y -45.308,Z -146.209,A -90.000,B 90.000,C 0.000} C_DIS
LIN {X 54.277,Y -45.308,Z -145.611,A -90.000,B 90.000,C 0.000} C_DIS
LIN {X 55.709,Y -45.308,Z -144.473,A -90.000,B 90.000,C 0.000} C_DIS
LIN {X 55.899,Y -45.308,Z -144.331,A -90.000,B 90.000,C 0.000} C_DIS
LIN {X 56.909,Y -45.308,Z -143.659,A -90.000,B 90.000,C 0.000} C_DIS
LIN {X 57.502,Y -45.308,Z -143.196,A -90.000,B 90.000,C 0.000} C_DIS
LIN {X 57.692,Y -45.308,Z -143.054,A -90.000,B 90.000,C 0.000} C_DIS
